REGION Network 4: Формирование событий линии
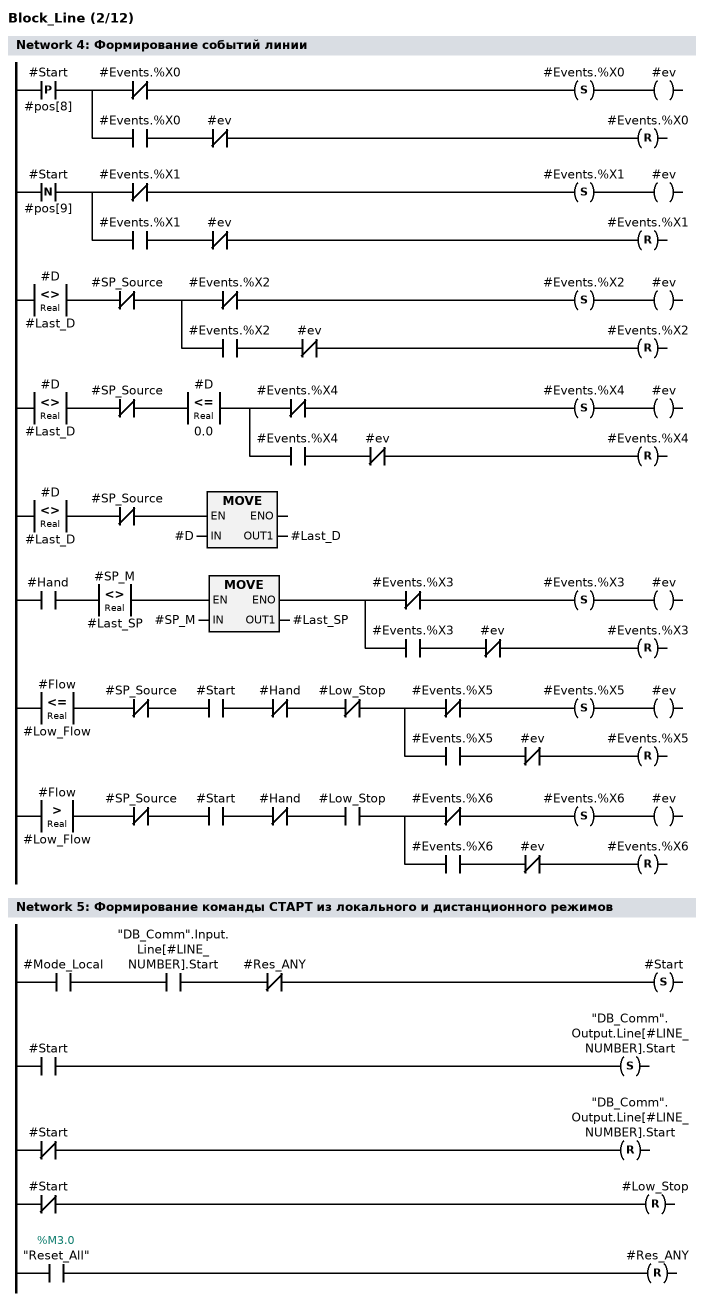
   RUNG wire#powerrail
      P_Contact(operand := #Start, bit := #pos[8])
      wire#w1
      I_Contact( #Events.%X0 )
      S_Coil( #Events.%X0 )
      Coil( #ev )
   END_RUNG
   RUNG wire#w1
      Contact( #Events.%X0 )
      I_Contact( #ev )
      R_Coil( #Events.%X0 )
   END_RUNG
   RUNG wire#powerrail
      N_Contact(operand := #Start, bit := #pos[9])
      wire#w2
      I_Contact( #Events.%X1 )
      S_Coil( #Events.%X1 )
      Coil( #ev )
   END_RUNG
   RUNG wire#w2
      Contact( #Events.%X1 )
      I_Contact( #ev )
      R_Coil( #Events.%X1 )
   END_RUNG
   RUNG wire#powerrail
      { S7_Templates := "SrcType := Real" } NE_Contact(in1 := #D, in2 := #Last_D)
      I_Contact( #SP_Source )
      wire#w3
      I_Contact( #Events.%X2 )
      S_Coil( #Events.%X2 )
      Coil( #ev )
   END_RUNG
   RUNG wire#w3
      Contact( #Events.%X2 )
      I_Contact( #ev )
      R_Coil( #Events.%X2 )
   END_RUNG
   RUNG wire#powerrail
      { S7_Templates := "SrcType := Real" } NE_Contact(in1 := #D, in2 := #Last_D)
      I_Contact( #SP_Source )
      { S7_Templates := "SrcType := Real" } LE_Contact(in1 := #D, in2 := 0.0)
      wire#w4
      I_Contact( #Events.%X4 )
      S_Coil( #Events.%X4 )
      Coil( #ev )
   END_RUNG
   RUNG wire#w4
      Contact( #Events.%X4 )
      I_Contact( #ev )
      R_Coil( #Events.%X4 )
   END_RUNG
   RUNG wire#powerrail
      { S7_Templates := "SrcType := Real" } NE_Contact(in1 := #D, in2 := #Last_D)
      I_Contact( #SP_Source )
      Move(in := #D, out1 => #Last_D)
   END_RUNG
   RUNG wire#powerrail
      Contact( #Hand )
      { S7_Templates := "SrcType := Real" } NE_Contact(in1 := #SP_M, in2 := #Last_SP)
      Move(in := #SP_M, out1 => #Last_SP)
      wire#w5
      I_Contact( #Events.%X3 )
      S_Coil( #Events.%X3 )
      Coil( #ev )
   END_RUNG
   RUNG wire#w5
      Contact( #Events.%X3 )
      I_Contact( #ev )
      R_Coil( #Events.%X3 )
   END_RUNG
   RUNG wire#powerrail
      { S7_Templates := "SrcType := Real" } LE_Contact(in1 := #Flow, in2 := #Low_Flow)
      I_Contact( #SP_Source )
      Contact( #Start )
      I_Contact( #Hand )
      I_Contact( #Low_Stop )
      wire#w6
      I_Contact( #Events.%X5 )
      S_Coil( #Events.%X5 )
      Coil( #ev )
   END_RUNG
   RUNG wire#w6
      Contact( #Events.%X5 )
      I_Contact( #ev )
      R_Coil( #Events.%X5 )
   END_RUNG
   RUNG wire#powerrail
      { S7_Templates := "SrcType := Real" } GT_Contact(in1 := #Flow, in2 := #Low_Flow)
      I_Contact( #SP_Source )
      Contact( #Start )
      I_Contact( #Hand )
      Contact( #Low_Stop )
      wire#w7
      I_Contact( #Events.%X6 )
      S_Coil( #Events.%X6 )
      Coil( #ev )
   END_RUNG
   RUNG wire#w7
      Contact( #Events.%X6 )
      I_Contact( #ev )
      R_Coil( #Events.%X6 )
   END_RUNG
   // the same network as SCL:
   #_w1 := #Start AND NOT #pos[8];   // rising edge of #Start
   #pos[8] := #Start;
   #_w2 := #_w1 AND NOT #Events.%X0;
   IF #_w2 THEN #Events.%X0 := TRUE; END_IF;
   #ev := #_w2;
   IF #_w1 AND #Events.%X0 AND NOT #ev THEN #Events.%X0 := FALSE; END_IF;
   #_w3 := NOT #Start AND #pos[9];   // falling edge of #Start
   #pos[9] := #Start;
   #_w4 := #_w3 AND NOT #Events.%X1;
   IF #_w4 THEN #Events.%X1 := TRUE; END_IF;
   #ev := #_w4;
   IF #_w3 AND #Events.%X1 AND NOT #ev THEN #Events.%X1 := FALSE; END_IF;
   #_w5 := (#D <> #Last_D) AND NOT #SP_Source;
   #_w6 := #_w5 AND NOT #Events.%X2;
   IF #_w6 THEN #Events.%X2 := TRUE; END_IF;
   #ev := #_w6;
   IF #_w5 AND #Events.%X2 AND NOT #ev THEN #Events.%X2 := FALSE; END_IF;
   #_w7 := (#D <> #Last_D) AND NOT #SP_Source AND (#D <= 0.0);
   #_w8 := #_w7 AND NOT #Events.%X4;
   IF #_w8 THEN #Events.%X4 := TRUE; END_IF;
   #ev := #_w8;
   IF #_w7 AND #Events.%X4 AND NOT #ev THEN #Events.%X4 := FALSE; END_IF;
   IF (#D <> #Last_D) AND NOT #SP_Source THEN #Last_D := #D; END_IF;
   #_w9 := #Hand AND (#SP_M <> #Last_SP);
   IF #_w9 THEN #Last_SP := #SP_M; END_IF;
   #_w10 := #_w9 AND NOT #Events.%X3;
   IF #_w10 THEN #Events.%X3 := TRUE; END_IF;
   #ev := #_w10;
   IF #_w9 AND #Events.%X3 AND NOT #ev THEN #Events.%X3 := FALSE; END_IF;
   #_w11 := (#Flow <= #Low_Flow) AND NOT #SP_Source AND #Start AND NOT #Hand AND NOT #Low_Stop;
   #_w12 := #_w11 AND NOT #Events.%X5;
   IF #_w12 THEN #Events.%X5 := TRUE; END_IF;
   #ev := #_w12;
   IF #_w11 AND #Events.%X5 AND NOT #ev THEN #Events.%X5 := FALSE; END_IF;
   #_w13 := (#Flow > #Low_Flow) AND NOT #SP_Source AND #Start AND NOT #Hand AND #Low_Stop;
   #_w14 := #_w13 AND NOT #Events.%X6;
   IF #_w14 THEN #Events.%X6 := TRUE; END_IF;
   #ev := #_w14;
   IF #_w13 AND #Events.%X6 AND NOT #ev THEN #Events.%X6 := FALSE; END_IF;
END_REGION

REGION Network 5: Формирование команды СТАРТ из локального и дистанционного режимов
   RUNG wire#powerrail
      Contact( #Mode_Local )
      Contact( "DB_Comm".Input.Line[#LINE_NUMBER].Start )
      I_Contact( #Res_ANY )
      S_Coil( #Start )
   END_RUNG
   RUNG wire#powerrail
      Contact( #Start )
      S_Coil( "DB_Comm".Output.Line[#LINE_NUMBER].Start )
   END_RUNG
   RUNG wire#powerrail
      I_Contact( #Start )
      R_Coil( "DB_Comm".Output.Line[#LINE_NUMBER].Start )
   END_RUNG
   RUNG wire#powerrail
      I_Contact( #Start )
      R_Coil( #Low_Stop )
   END_RUNG
   RUNG wire#powerrail
      Contact( "Reset_All" )
      R_Coil( #Res_ANY )
   END_RUNG
   // the same network as SCL:
   IF #Mode_Local AND "DB_Comm".Input.Line[#LINE_NUMBER].Start AND NOT #Res_ANY THEN #Start := TRUE; END_IF;
   IF #Start THEN "DB_Comm".Output.Line[#LINE_NUMBER].Start := TRUE; END_IF;
   IF NOT #Start THEN
       "DB_Comm".Output.Line[#LINE_NUMBER].Start := FALSE;
       #Low_Stop := FALSE;
   END_IF;
   IF "Reset_All" THEN #Res_ANY := FALSE; END_IF;
END_REGION

REGION Network 6: Старт - выбора насоса
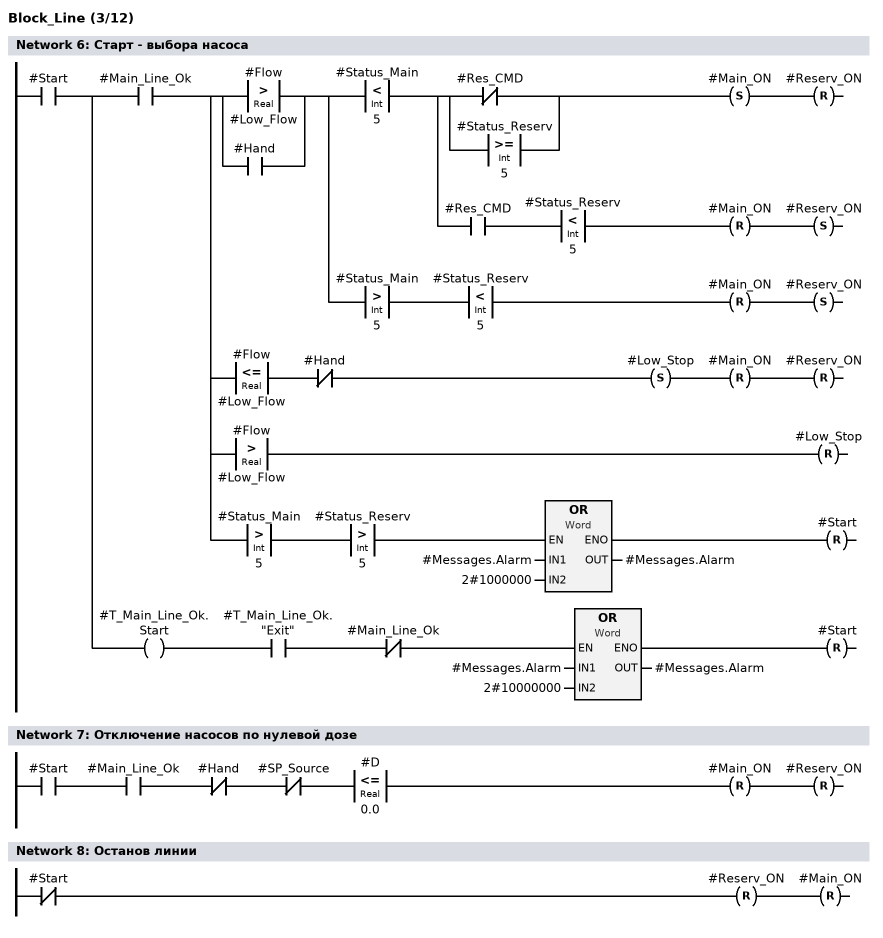
   #_w1 := #Start AND #Main_Line_Ok;
   #_w2 := #_w1 AND ((#Flow > #Low_Flow) OR #Hand);
   #_w3 := #_w2 AND (#Status_Main < 5);
   IF #_w3 AND (NOT #Res_CMD OR (#Status_Reserv >= 5)) THEN
       #Main_ON := TRUE;
       #Reserv_ON := FALSE;
   END_IF;
   IF #_w3 AND #Res_CMD AND (#Status_Reserv < 5) THEN
       #Main_ON := FALSE;
       #Reserv_ON := TRUE;
   END_IF;
   IF #_w2 AND (#Status_Main > 5) AND (#Status_Reserv < 5) THEN
       #Main_ON := FALSE;
       #Reserv_ON := TRUE;
   END_IF;
   IF #_w1 AND (#Flow <= #Low_Flow) AND NOT #Hand THEN
       #Low_Stop := TRUE;
       #Main_ON := FALSE;
       #Reserv_ON := FALSE;
   END_IF;
   IF #_w1 AND (#Flow > #Low_Flow) THEN #Low_Stop := FALSE; END_IF;
   IF #_w1 AND (#Status_Main > 5) AND (#Status_Reserv > 5) THEN
       #Messages.Alarm := #Messages.Alarm OR 2#1000000;
   END_IF;
   #_w4 := #Start;
   IF #_w1 AND (#Status_Main > 5) AND (#Status_Reserv > 5) THEN #Start := FALSE; END_IF;
   #T_Main_Line_Ok.Start := #_w4;
   IF #_w4 AND #T_Main_Line_Ok."Exit" AND NOT #Main_Line_Ok THEN
       #Messages.Alarm := #Messages.Alarm OR 2#10000000;
       #Start := FALSE;
   END_IF;
END_REGION

REGION Network 7: Отключение насосов по нулевой дозе
   RUNG wire#powerrail
      Contact( #Start )
      Contact( #Main_Line_Ok )
      I_Contact( #Hand )
      I_Contact( #SP_Source )
      { S7_Templates := "SrcType := Real" } LE_Contact(in1 := #D, in2 := 0.0)
      R_Coil( #Main_ON )
      R_Coil( #Reserv_ON )
   END_RUNG
   // the same network as SCL:
   IF #Start AND #Main_Line_Ok AND NOT #Hand AND NOT #SP_Source AND (#D <= 0.0) THEN
       #Main_ON := FALSE;
       #Reserv_ON := FALSE;
   END_IF;
END_REGION

REGION Network 8: Останов линии
   RUNG wire#powerrail
      I_Contact( #Start )
      R_Coil( #Reserv_ON )
      R_Coil( #Main_ON )
   END_RUNG
   // the same network as SCL:
   IF NOT #Start THEN
       #Reserv_ON := FALSE;
       #Main_ON := FALSE;
   END_IF;
END_REGION

REGION Network 9: Подсчёт наработки насосов и управление выбором основного и резервного
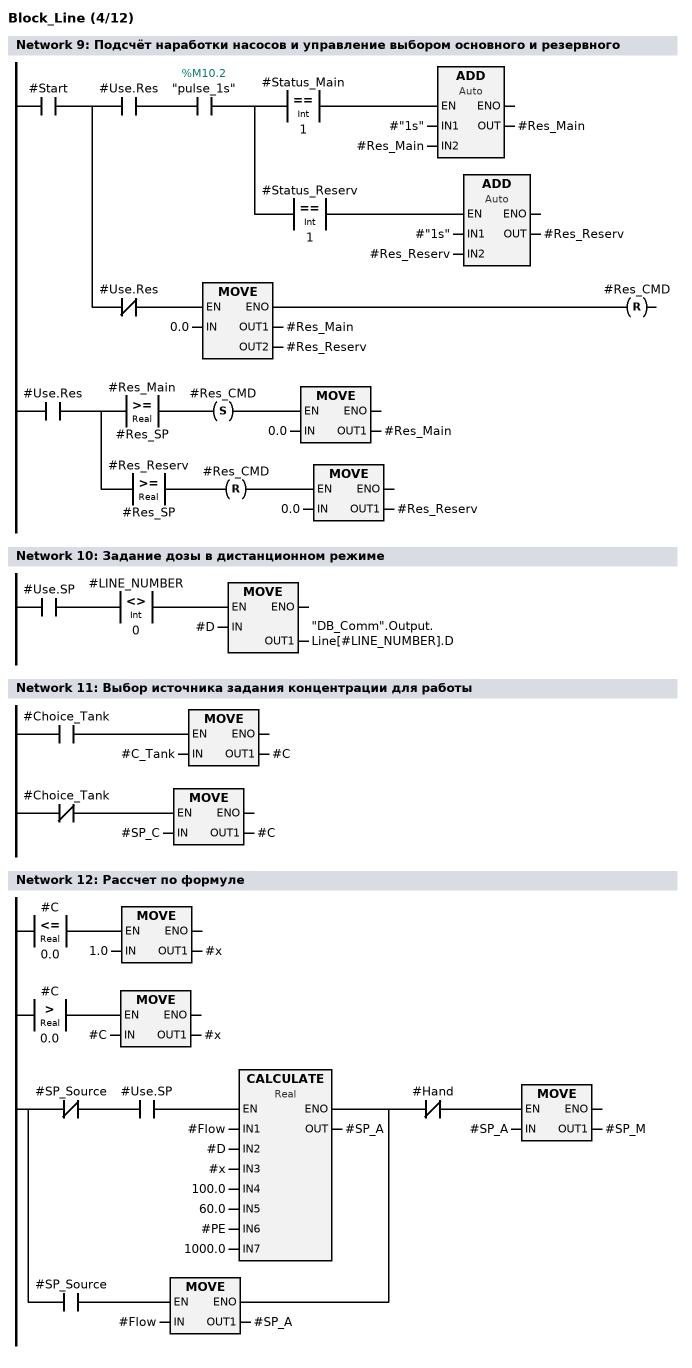
   RUNG wire#powerrail
      Contact( #Start )
      wire#w1
      Contact( #Use.Res )
      Contact( "pulse_1s" )
      wire#w2
      { S7_Templates := "SrcType := Int" } EQ_Contact(in1 := #Status_Main, in2 := 1)
      Add(in1 := #"1s", in2 := #Res_Main, out => #Res_Main)
   END_RUNG
   RUNG wire#w2
      { S7_Templates := "SrcType := Int" } EQ_Contact(in1 := #Status_Reserv, in2 := 1)
      Add(in1 := #"1s", in2 := #Res_Reserv, out => #Res_Reserv)
   END_RUNG
   RUNG wire#w1
      I_Contact( #Use.Res )
      Move(in := 0.0, out1 => #Res_Main, out2 => #Res_Reserv)
      R_Coil( #Res_CMD )
   END_RUNG
   RUNG wire#powerrail
      Contact( #Use.Res )
      wire#w3
      { S7_Templates := "SrcType := Real" } GE_Contact(in1 := #Res_Main, in2 := #Res_SP)
      S_Coil( #Res_CMD )
      Move(in := 0.0, out1 => #Res_Main)
   END_RUNG
   RUNG wire#w3
      { S7_Templates := "SrcType := Real" } GE_Contact(in1 := #Res_Reserv, in2 := #Res_SP)
      R_Coil( #Res_CMD )
      Move(in := 0.0, out1 => #Res_Reserv)
   END_RUNG
   // the same network as SCL:
   #_w1 := #Start AND #Use.Res AND "pulse_1s";
   IF #_w1 AND (#Status_Main = 1) THEN #Res_Main := #"1s" + #Res_Main; END_IF;
   IF #_w1 AND (#Status_Reserv = 1) THEN #Res_Reserv := #"1s" + #Res_Reserv; END_IF;
   IF #Start AND NOT #Use.Res THEN
       #Res_Main := 0.0;
       #Res_Reserv := 0.0;
       #Res_CMD := FALSE;
   END_IF;
   IF #Use.Res AND (#Res_Main >= #Res_SP) THEN
       #Res_CMD := TRUE;
       #Res_Main := 0.0;
   END_IF;
   IF #Use.Res AND (#Res_Reserv >= #Res_SP) THEN
       #Res_CMD := FALSE;
       #Res_Reserv := 0.0;
   END_IF;
END_REGION

REGION Network 10: Задание дозы в дистанционном режиме
   RUNG wire#powerrail
      Contact( #Use.SP )
      { S7_Templates := "SrcType := Int" } NE_Contact(in1 := #LINE_NUMBER, in2 := 0)
      Move(in := #D, out1 => "DB_Comm".Output.Line[#LINE_NUMBER].D)
   END_RUNG
   // the same network as SCL:
   IF #Use.SP AND (#LINE_NUMBER <> 0) THEN "DB_Comm".Output.Line[#LINE_NUMBER].D := #D; END_IF;
END_REGION

REGION Network 11: Выбор источника задания концентрации для работы
   RUNG wire#powerrail
      Contact( #Choice_Tank )
      Move(in := #C_Tank, out1 => #C)
   END_RUNG
   RUNG wire#powerrail
      I_Contact( #Choice_Tank )
      Move(in := #SP_C, out1 => #C)
   END_RUNG
   // the same network as SCL:
   IF #Choice_Tank THEN #C := #C_Tank; END_IF;
   IF NOT #Choice_Tank THEN #C := #SP_C; END_IF;
END_REGION

REGION Network 12: Рассчет по формуле
   RUNG wire#powerrail
      { S7_Templates := "SrcType := Real" } LE_Contact(in1 := #C, in2 := 0.0)
      Move(in := 1.0, out1 => #x)
   END_RUNG
   RUNG wire#powerrail
      { S7_Templates := "SrcType := Real" } GT_Contact(in1 := #C, in2 := 0.0)
      Move(in := #C, out1 => #x)
   END_RUNG
   RUNG wire#powerrail
      I_Contact( #SP_Source )
      Contact( #Use.SP )
      { S7_Templates := "SrcType := Real"; S7_Expression := "(IN2 * IN1) / ( IN3 / IN4) / (IN6 * IN7) / IN5" } Calculate(in1 := #Flow, in2 := #D, in3 := #x, in4 := 100.0, in5 := 60.0, in6 := #PE, in7 := 1000.0, out => #SP_A)
      wire#w1
      I_Contact( #Hand )
      Move(in := #SP_A, out1 => #SP_M)
   END_RUNG
   RUNG wire#powerrail
      Contact( #SP_Source )
      Move(in := #Flow, out1 => #SP_A)
   END_RUNG wire#w1
   // the same network as SCL:
   IF #C <= 0.0 THEN #x := 1.0; END_IF;
   IF #C > 0.0 THEN #x := #C; END_IF;
   #_w1 := NOT #SP_Source AND #Use.SP;
   IF #_w1 THEN #SP_A := (#D * #Flow) / ( #x / 100.0) / (#PE * 1000.0) / 60.0; END_IF;
   IF #SP_Source THEN #SP_A := #Flow; END_IF;
   IF (#_w1 OR #SP_Source) AND NOT #Hand THEN #SP_M := #SP_A; END_IF;
END_REGION

REGION Network 13: Выбор режима с разбавлением или без разбавления в дистанционном режиме
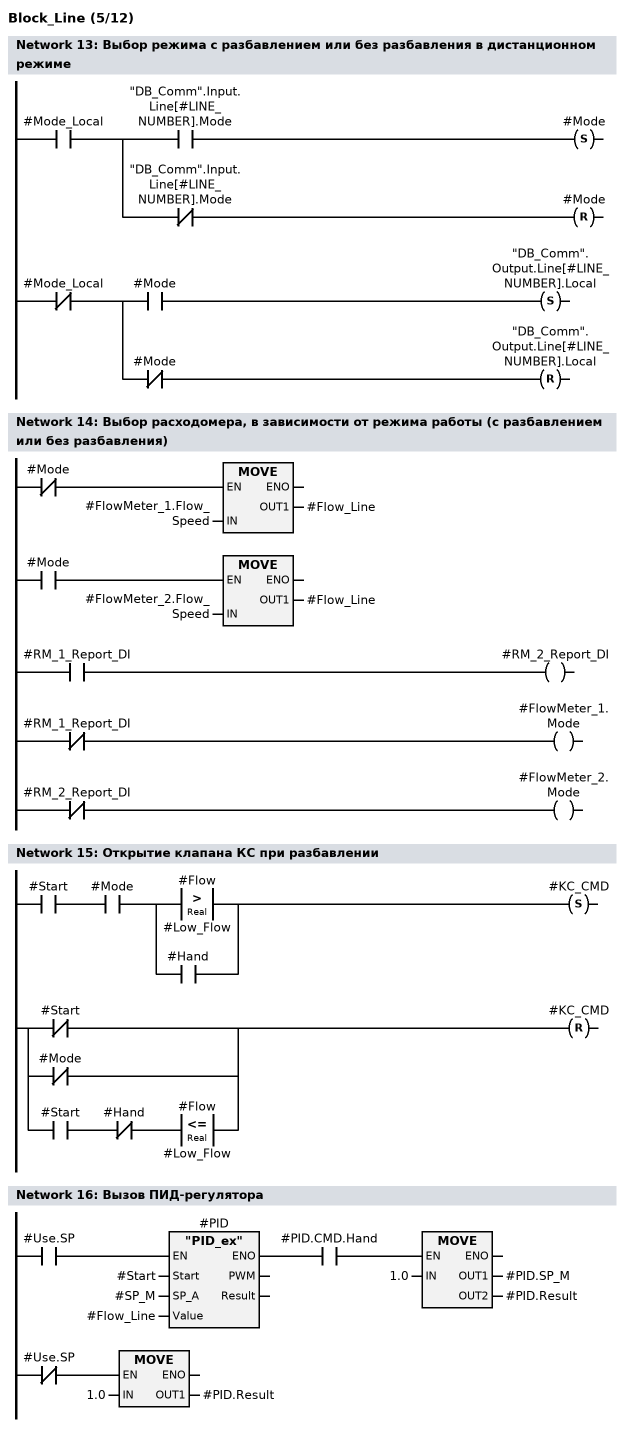
   RUNG wire#powerrail
      Contact( #Mode_Local )
      wire#w1
      Contact( "DB_Comm".Input.Line[#LINE_NUMBER].Mode )
      S_Coil( #Mode )
   END_RUNG
   RUNG wire#w1
      I_Contact( "DB_Comm".Input.Line[#LINE_NUMBER].Mode )
      R_Coil( #Mode )
   END_RUNG
   RUNG wire#powerrail
      I_Contact( #Mode_Local )
      wire#w2
      Contact( #Mode )
      S_Coil( "DB_Comm".Output.Line[#LINE_NUMBER].Local )
   END_RUNG
   RUNG wire#w2
      I_Contact( #Mode )
      R_Coil( "DB_Comm".Output.Line[#LINE_NUMBER].Local )
   END_RUNG
   // the same network as SCL:
   IF #Mode_Local AND "DB_Comm".Input.Line[#LINE_NUMBER].Mode THEN #Mode := TRUE; END_IF;
   IF #Mode_Local AND NOT "DB_Comm".Input.Line[#LINE_NUMBER].Mode THEN #Mode := FALSE; END_IF;
   IF NOT #Mode_Local AND #Mode THEN "DB_Comm".Output.Line[#LINE_NUMBER].Local := TRUE; END_IF;
   IF NOT #Mode_Local AND NOT #Mode THEN "DB_Comm".Output.Line[#LINE_NUMBER].Local := FALSE; END_IF;
END_REGION

REGION Network 14: Выбор расходомера, в зависимости от режима работы (с разбавлением или без разбавления)
   RUNG wire#powerrail
      I_Contact( #Mode )
      Move(in := #FlowMeter_1.Flow_Speed, out1 => #Flow_Line)
   END_RUNG
   RUNG wire#powerrail
      Contact( #Mode )
      Move(in := #FlowMeter_2.Flow_Speed, out1 => #Flow_Line)
   END_RUNG
   RUNG wire#powerrail
      Contact( #RM_1_Report_DI )
      Coil( #RM_2_Report_DI )
   END_RUNG
   RUNG wire#powerrail
      I_Contact( #RM_1_Report_DI )
      Coil( #FlowMeter_1.Mode )
   END_RUNG
   RUNG wire#powerrail
      I_Contact( #RM_2_Report_DI )
      Coil( #FlowMeter_2.Mode )
   END_RUNG
   // the same network as SCL:
   IF NOT #Mode THEN #Flow_Line := #FlowMeter_1.Flow_Speed; END_IF;
   IF #Mode THEN #Flow_Line := #FlowMeter_2.Flow_Speed; END_IF;
   #RM_2_Report_DI := #RM_1_Report_DI;
   #FlowMeter_1.Mode := NOT #RM_1_Report_DI;
   #FlowMeter_2.Mode := NOT #RM_2_Report_DI;
END_REGION

REGION Network 15: Открытие клапана КС при разбавлении
   RUNG wire#powerrail
      Contact( #Start )
      Contact( #Mode )
      wire#w1
      { S7_Templates := "SrcType := Real" } GT_Contact(in1 := #Flow, in2 := #Low_Flow)
      wire#w2
      S_Coil( #KC_CMD )
   END_RUNG
   RUNG wire#w1
      Contact( #Hand )
   END_RUNG wire#w2
   RUNG wire#powerrail
      I_Contact( #Start )
      wire#w3
      R_Coil( #KC_CMD )
   END_RUNG
   RUNG wire#powerrail
      I_Contact( #Mode )
   END_RUNG wire#w3
   RUNG wire#powerrail
      Contact( #Start )
      I_Contact( #Hand )
      { S7_Templates := "SrcType := Real" } LE_Contact(in1 := #Flow, in2 := #Low_Flow)
   END_RUNG wire#w3
   // the same network as SCL:
   IF #Start AND #Mode AND ((#Flow > #Low_Flow) OR #Hand) THEN #KC_CMD := TRUE; END_IF;
   IF NOT #Start OR NOT #Mode OR (#Start AND NOT #Hand AND (#Flow <= #Low_Flow)) THEN
       #KC_CMD := FALSE;
   END_IF;
END_REGION

REGION Network 16: Вызов ПИД-регулятора
   RUNG wire#powerrail
      Contact( #Use.SP )
      #PID(Start := #Start, SP_A := #SP_M, Value := #Flow_Line, PWM =>, Result =>)
      Contact( #PID.CMD.Hand )
      Move(in := 1.0, out1 => #PID.SP_M, out2 => #PID.Result)
   END_RUNG
   RUNG wire#powerrail
      I_Contact( #Use.SP )
      Move(in := 1.0, out1 => #PID.Result)
   END_RUNG
   // the same network as SCL:
   #PID(EN := #Use.SP, Start := #Start, SP_A := #SP_M, Value := #Flow_Line, ENO => #_w1);   // "PID_ex"
   IF #_w1 AND #PID.CMD.Hand THEN
       #PID.SP_M := 1.0;
       #PID.Result := 1.0;
   END_IF;
   IF NOT #Use.SP THEN #PID.Result := 1.0; END_IF;
END_REGION

REGION Network 17: Обнуление уставки при отстутствии аналогового управления насосами
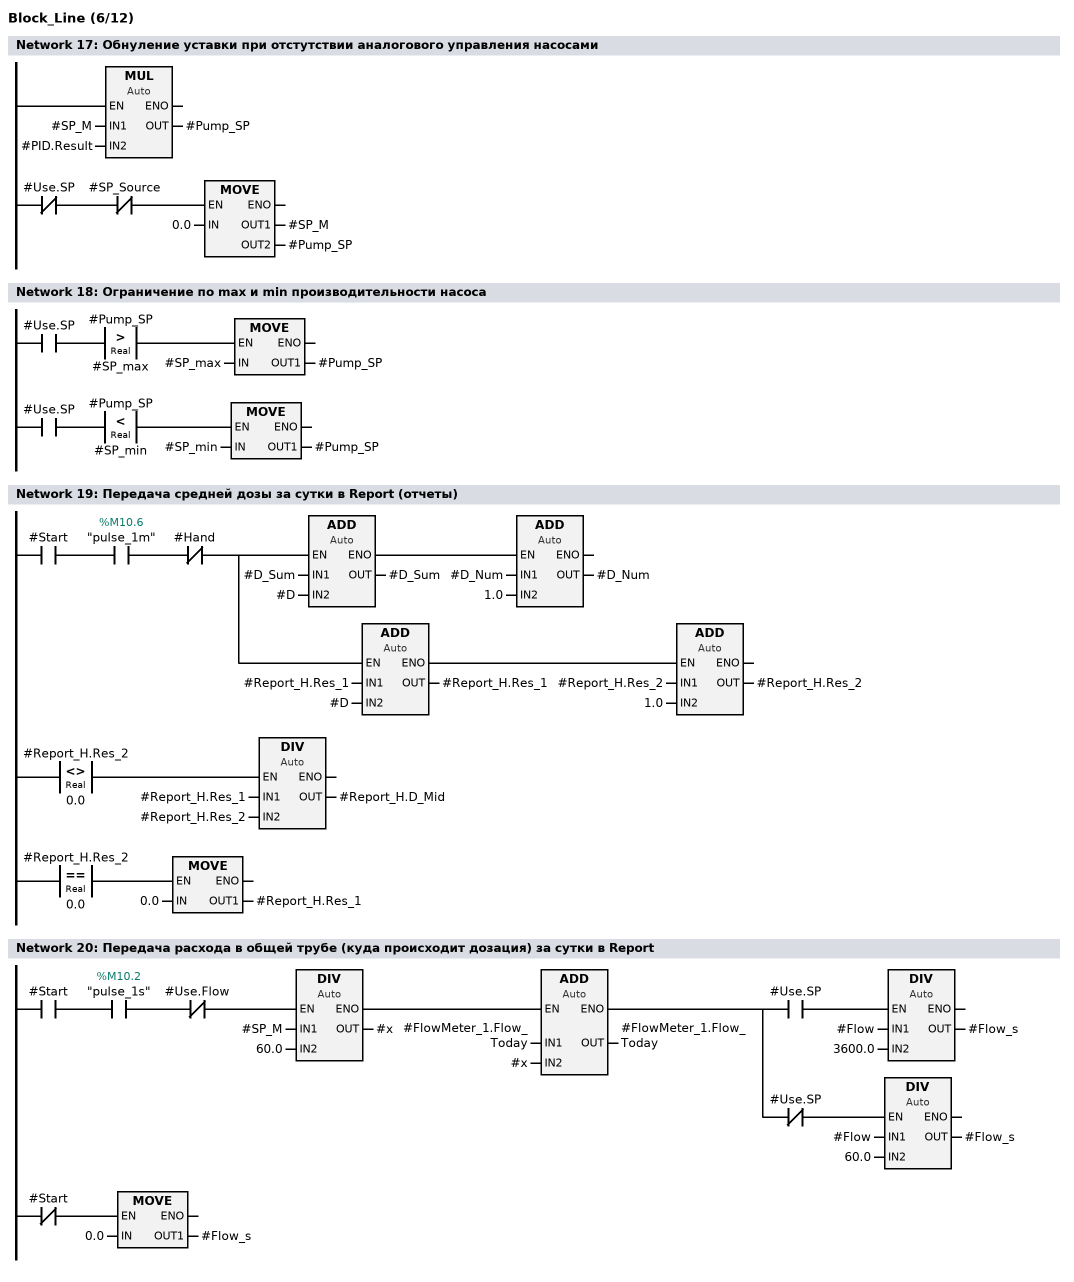
   RUNG wire#powerrail
      Mul(in1 := #SP_M, in2 := #PID.Result, out => #Pump_SP)
   END_RUNG
   RUNG wire#powerrail
      I_Contact( #Use.SP )
      I_Contact( #SP_Source )
      Move(in := 0.0, out1 => #SP_M, out2 => #Pump_SP)
   END_RUNG
   // the same network as SCL:
   #Pump_SP := #SP_M * #PID.Result;
   IF NOT #Use.SP AND NOT #SP_Source THEN
       #SP_M := 0.0;
       #Pump_SP := 0.0;
   END_IF;
END_REGION

REGION Network 18: Ограничение по max и min производительности насоса
   RUNG wire#powerrail
      Contact( #Use.SP )
      { S7_Templates := "SrcType := Real" } GT_Contact(in1 := #Pump_SP, in2 := #SP_max)
      Move(in := #SP_max, out1 => #Pump_SP)
   END_RUNG
   RUNG wire#powerrail
      Contact( #Use.SP )
      { S7_Templates := "SrcType := Real" } LT_Contact(in1 := #Pump_SP, in2 := #SP_min)
      Move(in := #SP_min, out1 => #Pump_SP)
   END_RUNG
   // the same network as SCL:
   IF #Use.SP AND (#Pump_SP > #SP_max) THEN #Pump_SP := #SP_max; END_IF;
   IF #Use.SP AND (#Pump_SP < #SP_min) THEN #Pump_SP := #SP_min; END_IF;
END_REGION

REGION Network 19: Передача средней дозы за сутки в Report (отчеты)
   RUNG wire#powerrail
      Contact( #Start )
      Contact( "pulse_1m" )
      I_Contact( #Hand )
      wire#w1
      Add(in1 := #D_Sum, in2 := #D, out => #D_Sum)
      Add(in1 := #D_Num, in2 := 1.0, out => #D_Num)
   END_RUNG
   RUNG wire#w1
      Add(in1 := #Report_H.Res_1, in2 := #D, out => #Report_H.Res_1)
      Add(in1 := #Report_H.Res_2, in2 := 1.0, out => #Report_H.Res_2)
   END_RUNG
   RUNG wire#powerrail
      { S7_Templates := "SrcType := Real" } NE_Contact(in1 := #Report_H.Res_2, in2 := 0.0)
      Div(in1 := #Report_H.Res_1, in2 := #Report_H.Res_2, out => #Report_H.D_Mid)
   END_RUNG
   RUNG wire#powerrail
      { S7_Templates := "SrcType := Real" } EQ_Contact(in1 := #Report_H.Res_2, in2 := 0.0)
      Move(in := 0.0, out1 => #Report_H.Res_1)
   END_RUNG
   // the same network as SCL:
   IF #Start AND "pulse_1m" AND NOT #Hand THEN
       #D_Sum := #D_Sum + #D;
       #D_Num := #D_Num + 1.0;
       #Report_H.Res_1 := #Report_H.Res_1 + #D;
       #Report_H.Res_2 := #Report_H.Res_2 + 1.0;
   END_IF;
   IF #Report_H.Res_2 <> 0.0 THEN #Report_H.D_Mid := #Report_H.Res_1 / #Report_H.Res_2; END_IF;
   IF #Report_H.Res_2 = 0.0 THEN #Report_H.Res_1 := 0.0; END_IF;
END_REGION

REGION Network 20: Передача расхода в общей трубе (куда происходит дозация) за сутки в Report
   RUNG wire#powerrail
      Contact( #Start )
      Contact( "pulse_1s" )
      I_Contact( #Use.Flow )
      Div(in1 := #SP_M, in2 := 60.0, out => #x)
      Add(in1 := #FlowMeter_1.Flow_Today, in2 := #x, out => #FlowMeter_1.Flow_Today)
      wire#w1
      Contact( #Use.SP )
      Div(in1 := #Flow, in2 := 3600.0, out => #Flow_s)
   END_RUNG
   RUNG wire#w1
      I_Contact( #Use.SP )
      Div(in1 := #Flow, in2 := 60.0, out => #Flow_s)
   END_RUNG
   RUNG wire#powerrail
      I_Contact( #Start )
      Move(in := 0.0, out1 => #Flow_s)
   END_RUNG
   // the same network as SCL:
   #_w1 := #Start AND "pulse_1s" AND NOT #Use.Flow;
   IF #_w1 THEN
       #x := #SP_M / 60.0;
       #FlowMeter_1.Flow_Today := #FlowMeter_1.Flow_Today + #x;
   END_IF;
   IF #_w1 AND #Use.SP THEN #Flow_s := #Flow / 3600.0; END_IF;
   IF #_w1 AND NOT #Use.SP THEN #Flow_s := #Flow / 60.0; END_IF;
   IF NOT #Start THEN #Flow_s := 0.0; END_IF;
END_REGION

REGION Network 21: Авария основного насоса по датчику протока
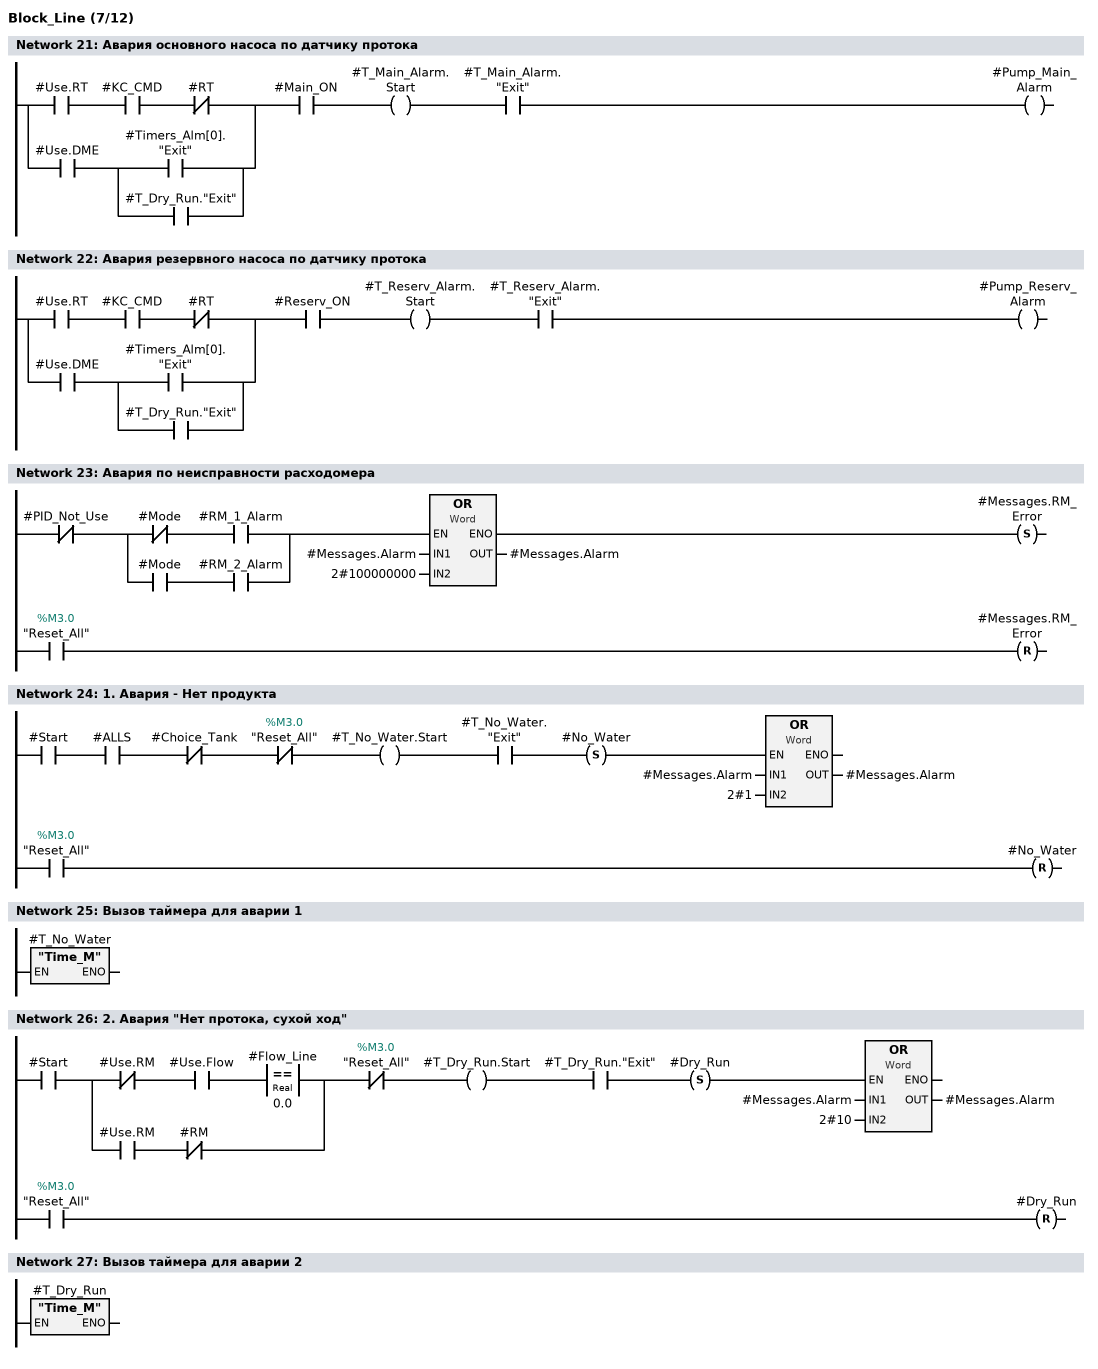
   RUNG wire#powerrail
      Contact( #Use.RT )
      Contact( #KC_CMD )
      I_Contact( #RT )
      wire#w1
      Contact( #Main_ON )
      Coil( #T_Main_Alarm.Start )
      Contact( #T_Main_Alarm."Exit" )
      Coil( #Pump_Main_Alarm )
   END_RUNG
   RUNG wire#powerrail
      Contact( #Use.DME )
      wire#w2
      Contact( #Timers_Alm[0]."Exit" )
   END_RUNG wire#w1
   RUNG wire#w2
      Contact( #T_Dry_Run."Exit" )
   END_RUNG wire#w1
   // the same network as SCL:
   #T_Main_Alarm.Start := ((#Use.RT AND #KC_CMD AND NOT #RT) OR (#Use.DME AND (#Timers_Alm[0]."Exit" OR #T_Dry_Run."Exit"))) AND #Main_ON;
   #Pump_Main_Alarm := #T_Main_Alarm.Start AND #T_Main_Alarm."Exit";
END_REGION

REGION Network 22: Авария резервного насоса по датчику протока
   RUNG wire#powerrail
      Contact( #Use.RT )
      Contact( #KC_CMD )
      I_Contact( #RT )
      wire#w1
      Contact( #Reserv_ON )
      Coil( #T_Reserv_Alarm.Start )
      Contact( #T_Reserv_Alarm."Exit" )
      Coil( #Pump_Reserv_Alarm )
   END_RUNG
   RUNG wire#powerrail
      Contact( #Use.DME )
      wire#w2
      Contact( #Timers_Alm[0]."Exit" )
   END_RUNG wire#w1
   RUNG wire#w2
      Contact( #T_Dry_Run."Exit" )
   END_RUNG wire#w1
   // the same network as SCL:
   #T_Reserv_Alarm.Start := ((#Use.RT AND #KC_CMD AND NOT #RT) OR (#Use.DME AND (#Timers_Alm[0]."Exit" OR #T_Dry_Run."Exit"))) AND #Reserv_ON;
   #Pump_Reserv_Alarm := #T_Reserv_Alarm.Start AND #T_Reserv_Alarm."Exit";
END_REGION

REGION Network 23: Авария по неисправности расходомера
   IF NOT #PID_Not_Use AND ((NOT #Mode AND #RM_1_Alarm) OR (#Mode AND #RM_2_Alarm)) THEN
       #Messages.Alarm := #Messages.Alarm OR 2#100000000;
       #Messages.RM_Error := TRUE;
   END_IF;
   IF "Reset_All" THEN #Messages.RM_Error := FALSE; END_IF;
END_REGION

REGION Network 24: 1. Авария - Нет продукта
   #T_No_Water.Start := #Start AND #ALLS AND NOT #Choice_Tank AND NOT "Reset_All";
   IF #T_No_Water.Start AND #T_No_Water."Exit" THEN
       #No_Water := TRUE;
       #Messages.Alarm := #Messages.Alarm OR 2#1;
   END_IF;
   IF "Reset_All" THEN #No_Water := FALSE; END_IF;
END_REGION

REGION Network 25: Вызов таймера для аварии 1
   RUNG wire#powerrail
      #T_No_Water()
   END_RUNG
   // the same network as SCL:
   #T_No_Water();   // "Time_M"
END_REGION

REGION Network 26: 2. Авария "Нет протока, сухой ход"
   #T_Dry_Run.Start := #Start AND ((NOT #Use.RM AND #Use.Flow AND (#Flow_Line = 0.0)) OR (#Use.RM AND NOT #RM)) AND NOT "Reset_All";
   IF #T_Dry_Run.Start AND #T_Dry_Run."Exit" THEN
       #Dry_Run := TRUE;
       #Messages.Alarm := #Messages.Alarm OR 2#10;
   END_IF;
   IF "Reset_All" THEN #Dry_Run := FALSE; END_IF;
END_REGION

REGION Network 27: Вызов таймера для аварии 2
   RUNG wire#powerrail
      #T_Dry_Run()
   END_RUNG
   // the same network as SCL:
   #T_Dry_Run();   // "Time_M"
END_REGION

REGION Network 28: 3. Авария - низкий проток
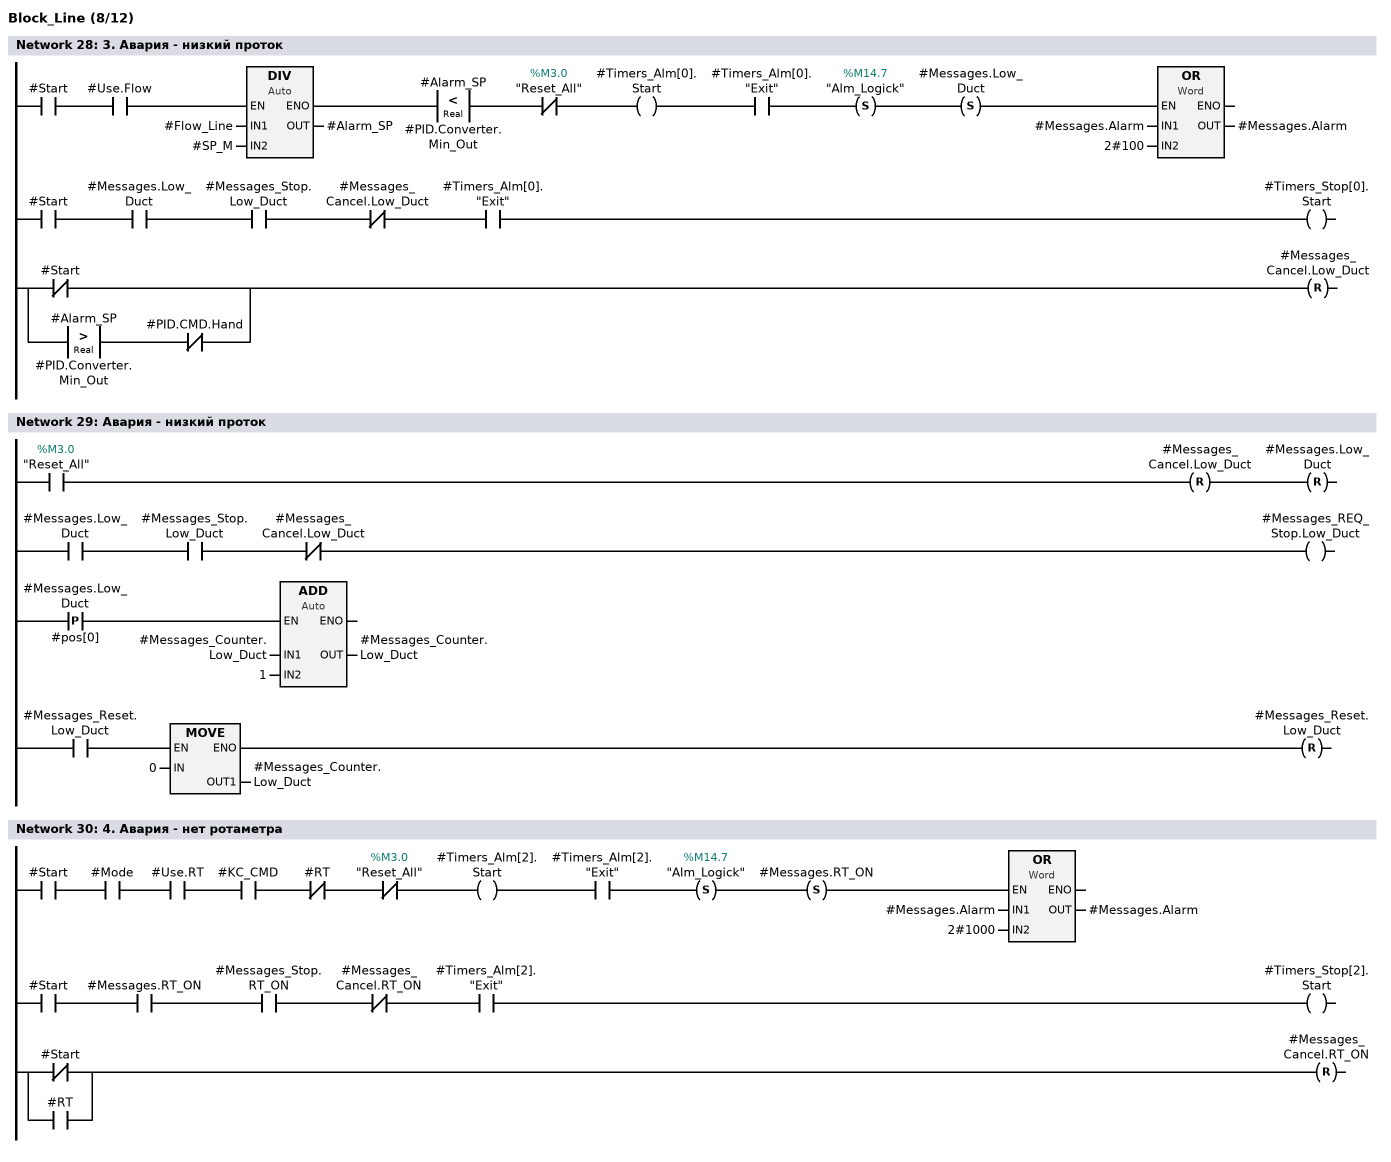
   #_w1 := #Start AND #Use.Flow;
   IF #_w1 THEN #Alarm_SP := #Flow_Line / #SP_M; END_IF;
   #Timers_Alm[0].Start := #_w1 AND (#Alarm_SP < #PID.Converter.Min_Out) AND NOT "Reset_All";
   IF #_w1 AND (#Alarm_SP < #PID.Converter.Min_Out) AND NOT "Reset_All" AND #Timers_Alm[0]."Exit" THEN
       "Alm_Logick" := TRUE;
       #Messages.Low_Duct := TRUE;
       #Messages.Alarm := #Messages.Alarm OR 2#100;
   END_IF;
   #Timers_Stop[0].Start := #Start AND #Messages.Low_Duct AND #Messages_Stop.Low_Duct AND NOT #Messages_Cancel.Low_Duct AND #Timers_Alm[0]."Exit";
   IF NOT #Start OR ((#Alarm_SP > #PID.Converter.Min_Out) AND NOT #PID.CMD.Hand) THEN
       #Messages_Cancel.Low_Duct := FALSE;
   END_IF;
END_REGION

REGION Network 29: Авария - низкий проток
   RUNG wire#powerrail
      Contact( "Reset_All" )
      R_Coil( #Messages_Cancel.Low_Duct )
      R_Coil( #Messages.Low_Duct )
   END_RUNG
   RUNG wire#powerrail
      Contact( #Messages.Low_Duct )
      Contact( #Messages_Stop.Low_Duct )
      I_Contact( #Messages_Cancel.Low_Duct )
      Coil( #Messages_REQ_Stop.Low_Duct )
   END_RUNG
   RUNG wire#powerrail
      P_Contact(operand := #Messages.Low_Duct, bit := #pos[0])
      Add(in1 := #Messages_Counter.Low_Duct, in2 := 1, out => #Messages_Counter.Low_Duct)
   END_RUNG
   RUNG wire#powerrail
      Contact( #Messages_Reset.Low_Duct )
      Move(in := 0, out1 => #Messages_Counter.Low_Duct)
      R_Coil( #Messages_Reset.Low_Duct )
   END_RUNG
   // the same network as SCL:
   IF "Reset_All" THEN
       #Messages_Cancel.Low_Duct := FALSE;
       #Messages.Low_Duct := FALSE;
   END_IF;
   #Messages_REQ_Stop.Low_Duct := #Messages.Low_Duct AND #Messages_Stop.Low_Duct AND NOT #Messages_Cancel.Low_Duct;
   #_w1 := #Messages.Low_Duct AND NOT #pos[0];   // rising edge of #Messages.Low_Duct
   #pos[0] := #Messages.Low_Duct;
   IF #_w1 THEN #Messages_Counter.Low_Duct := #Messages_Counter.Low_Duct + 1; END_IF;
   IF #Messages_Reset.Low_Duct THEN
       #Messages_Counter.Low_Duct := 0;
       #Messages_Reset.Low_Duct := FALSE;
   END_IF;
END_REGION

REGION Network 30: 4. Авария - нет ротаметра
   #Timers_Alm[2].Start := #Start AND #Mode AND #Use.RT AND #KC_CMD AND NOT #RT AND NOT "Reset_All";
   IF #Start AND #Mode AND #Use.RT AND #KC_CMD AND NOT #RT AND NOT "Reset_All" AND #Timers_Alm[2]."Exit" THEN
       "Alm_Logick" := TRUE;
       #Messages.RT_ON := TRUE;
       #Messages.Alarm := #Messages.Alarm OR 2#1000;
   END_IF;
   #Timers_Stop[2].Start := #Start AND #Messages.RT_ON AND #Messages_Stop.RT_ON AND NOT #Messages_Cancel.RT_ON AND #Timers_Alm[2]."Exit";
   IF NOT #Start OR #RT THEN #Messages_Cancel.RT_ON := FALSE; END_IF;
END_REGION

REGION Network 31: Авария - нет ротаметра
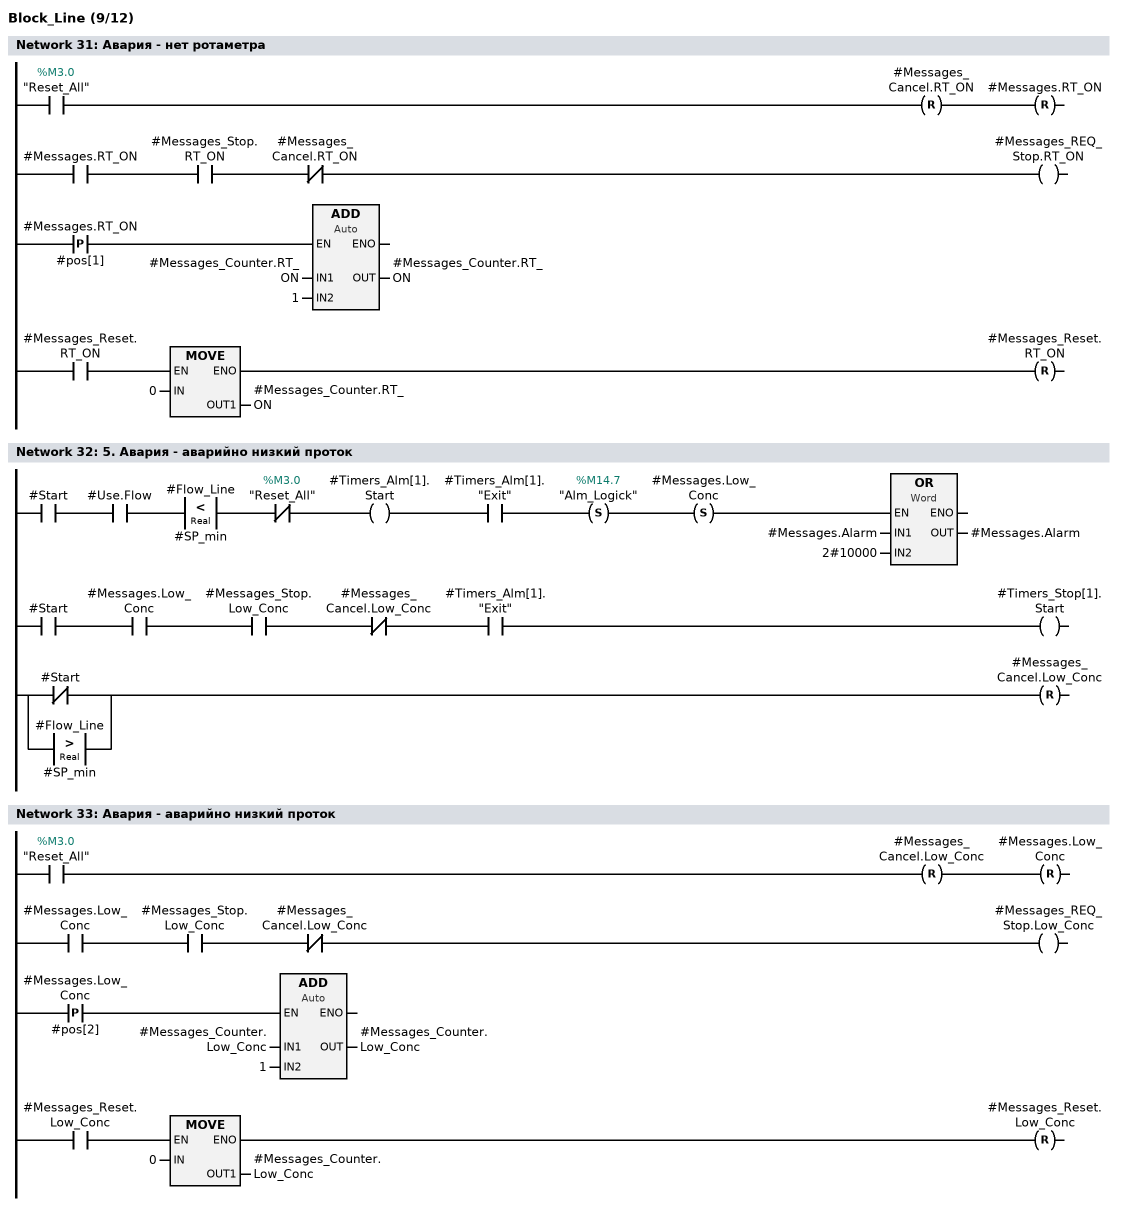
   RUNG wire#powerrail
      Contact( "Reset_All" )
      R_Coil( #Messages_Cancel.RT_ON )
      R_Coil( #Messages.RT_ON )
   END_RUNG
   RUNG wire#powerrail
      Contact( #Messages.RT_ON )
      Contact( #Messages_Stop.RT_ON )
      I_Contact( #Messages_Cancel.RT_ON )
      Coil( #Messages_REQ_Stop.RT_ON )
   END_RUNG
   RUNG wire#powerrail
      P_Contact(operand := #Messages.RT_ON, bit := #pos[1])
      Add(in1 := #Messages_Counter.RT_ON, in2 := 1, out => #Messages_Counter.RT_ON)
   END_RUNG
   RUNG wire#powerrail
      Contact( #Messages_Reset.RT_ON )
      Move(in := 0, out1 => #Messages_Counter.RT_ON)
      R_Coil( #Messages_Reset.RT_ON )
   END_RUNG
   // the same network as SCL:
   IF "Reset_All" THEN
       #Messages_Cancel.RT_ON := FALSE;
       #Messages.RT_ON := FALSE;
   END_IF;
   #Messages_REQ_Stop.RT_ON := #Messages.RT_ON AND #Messages_Stop.RT_ON AND NOT #Messages_Cancel.RT_ON;
   #_w1 := #Messages.RT_ON AND NOT #pos[1];   // rising edge of #Messages.RT_ON
   #pos[1] := #Messages.RT_ON;
   IF #_w1 THEN #Messages_Counter.RT_ON := #Messages_Counter.RT_ON + 1; END_IF;
   IF #Messages_Reset.RT_ON THEN
       #Messages_Counter.RT_ON := 0;
       #Messages_Reset.RT_ON := FALSE;
   END_IF;
END_REGION

REGION Network 32: 5. Авария - аварийно низкий проток
   #Timers_Alm[1].Start := #Start AND #Use.Flow AND (#Flow_Line < #SP_min) AND NOT "Reset_All";
   IF #Start AND #Use.Flow AND (#Flow_Line < #SP_min) AND NOT "Reset_All" AND #Timers_Alm[1]."Exit" THEN
       "Alm_Logick" := TRUE;
       #Messages.Low_Conc := TRUE;
       #Messages.Alarm := #Messages.Alarm OR 2#10000;
   END_IF;
   #Timers_Stop[1].Start := #Start AND #Messages.Low_Conc AND #Messages_Stop.Low_Conc AND NOT #Messages_Cancel.Low_Conc AND #Timers_Alm[1]."Exit";
   IF NOT #Start OR (#Flow_Line > #SP_min) THEN #Messages_Cancel.Low_Conc := FALSE; END_IF;
END_REGION

REGION Network 33: Авария - аварийно низкий проток
   RUNG wire#powerrail
      Contact( "Reset_All" )
      R_Coil( #Messages_Cancel.Low_Conc )
      R_Coil( #Messages.Low_Conc )
   END_RUNG
   RUNG wire#powerrail
      Contact( #Messages.Low_Conc )
      Contact( #Messages_Stop.Low_Conc )
      I_Contact( #Messages_Cancel.Low_Conc )
      Coil( #Messages_REQ_Stop.Low_Conc )
   END_RUNG
   RUNG wire#powerrail
      P_Contact(operand := #Messages.Low_Conc, bit := #pos[2])
      Add(in1 := #Messages_Counter.Low_Conc, in2 := 1, out => #Messages_Counter.Low_Conc)
   END_RUNG
   RUNG wire#powerrail
      Contact( #Messages_Reset.Low_Conc )
      Move(in := 0, out1 => #Messages_Counter.Low_Conc)
      R_Coil( #Messages_Reset.Low_Conc )
   END_RUNG
   // the same network as SCL:
   IF "Reset_All" THEN
       #Messages_Cancel.Low_Conc := FALSE;
       #Messages.Low_Conc := FALSE;
   END_IF;
   #Messages_REQ_Stop.Low_Conc := #Messages.Low_Conc AND #Messages_Stop.Low_Conc AND NOT #Messages_Cancel.Low_Conc;
   #_w1 := #Messages.Low_Conc AND NOT #pos[2];   // rising edge of #Messages.Low_Conc
   #pos[2] := #Messages.Low_Conc;
   IF #_w1 THEN #Messages_Counter.Low_Conc := #Messages_Counter.Low_Conc + 1; END_IF;
   IF #Messages_Reset.Low_Conc THEN
       #Messages_Counter.Low_Conc := 0;
       #Messages_Reset.Low_Conc := FALSE;
   END_IF;
END_REGION

REGION Network 34: 6. Авария - застрял ротаметр
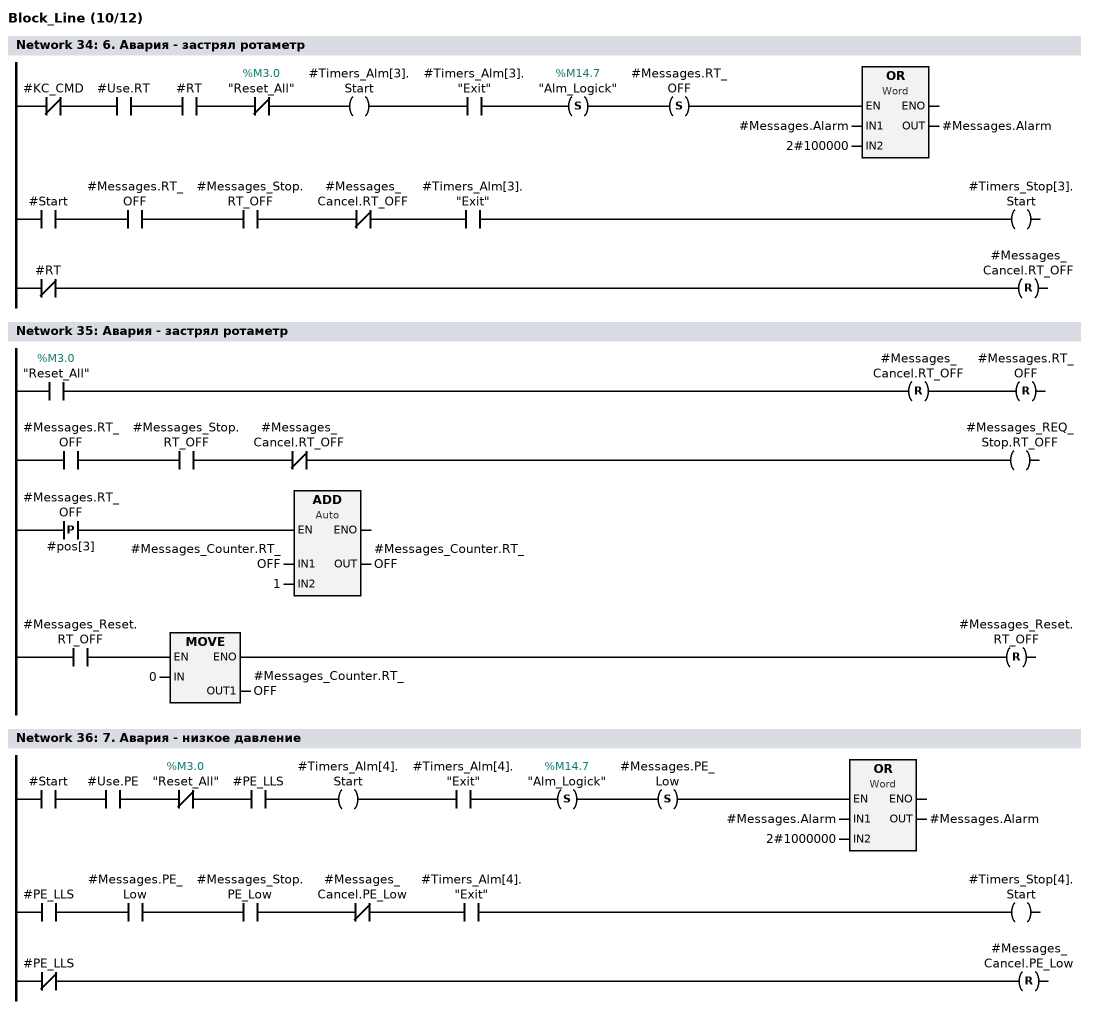
   #Timers_Alm[3].Start := NOT #KC_CMD AND #Use.RT AND #RT AND NOT "Reset_All";
   IF NOT #KC_CMD AND #Use.RT AND #RT AND NOT "Reset_All" AND #Timers_Alm[3]."Exit" THEN
       "Alm_Logick" := TRUE;
       #Messages.RT_OFF := TRUE;
       #Messages.Alarm := #Messages.Alarm OR 2#100000;
   END_IF;
   #Timers_Stop[3].Start := #Start AND #Messages.RT_OFF AND #Messages_Stop.RT_OFF AND NOT #Messages_Cancel.RT_OFF AND #Timers_Alm[3]."Exit";
   IF NOT #RT THEN #Messages_Cancel.RT_OFF := FALSE; END_IF;
END_REGION

REGION Network 35: Авария - застрял ротаметр
   RUNG wire#powerrail
      Contact( "Reset_All" )
      R_Coil( #Messages_Cancel.RT_OFF )
      R_Coil( #Messages.RT_OFF )
   END_RUNG
   RUNG wire#powerrail
      Contact( #Messages.RT_OFF )
      Contact( #Messages_Stop.RT_OFF )
      I_Contact( #Messages_Cancel.RT_OFF )
      Coil( #Messages_REQ_Stop.RT_OFF )
   END_RUNG
   RUNG wire#powerrail
      P_Contact(operand := #Messages.RT_OFF, bit := #pos[3])
      Add(in1 := #Messages_Counter.RT_OFF, in2 := 1, out => #Messages_Counter.RT_OFF)
   END_RUNG
   RUNG wire#powerrail
      Contact( #Messages_Reset.RT_OFF )
      Move(in := 0, out1 => #Messages_Counter.RT_OFF)
      R_Coil( #Messages_Reset.RT_OFF )
   END_RUNG
   // the same network as SCL:
   IF "Reset_All" THEN
       #Messages_Cancel.RT_OFF := FALSE;
       #Messages.RT_OFF := FALSE;
   END_IF;
   #Messages_REQ_Stop.RT_OFF := #Messages.RT_OFF AND #Messages_Stop.RT_OFF AND NOT #Messages_Cancel.RT_OFF;
   #_w1 := #Messages.RT_OFF AND NOT #pos[3];   // rising edge of #Messages.RT_OFF
   #pos[3] := #Messages.RT_OFF;
   IF #_w1 THEN #Messages_Counter.RT_OFF := #Messages_Counter.RT_OFF + 1; END_IF;
   IF #Messages_Reset.RT_OFF THEN
       #Messages_Counter.RT_OFF := 0;
       #Messages_Reset.RT_OFF := FALSE;
   END_IF;
END_REGION

REGION Network 36: 7. Авария - низкое давление
   #Timers_Alm[4].Start := #Start AND #Use.PE AND NOT "Reset_All" AND #PE_LLS;
   IF #Start AND #Use.PE AND NOT "Reset_All" AND #PE_LLS AND #Timers_Alm[4]."Exit" THEN
       "Alm_Logick" := TRUE;
       #Messages.PE_Low := TRUE;
       #Messages.Alarm := #Messages.Alarm OR 2#1000000;
   END_IF;
   #Timers_Stop[4].Start := #PE_LLS AND #Messages.PE_Low AND #Messages_Stop.PE_Low AND NOT #Messages_Cancel.PE_Low AND #Timers_Alm[4]."Exit";
   IF NOT #PE_LLS THEN #Messages_Cancel.PE_Low := FALSE; END_IF;
END_REGION

REGION Network 37: Авария - низкое давление
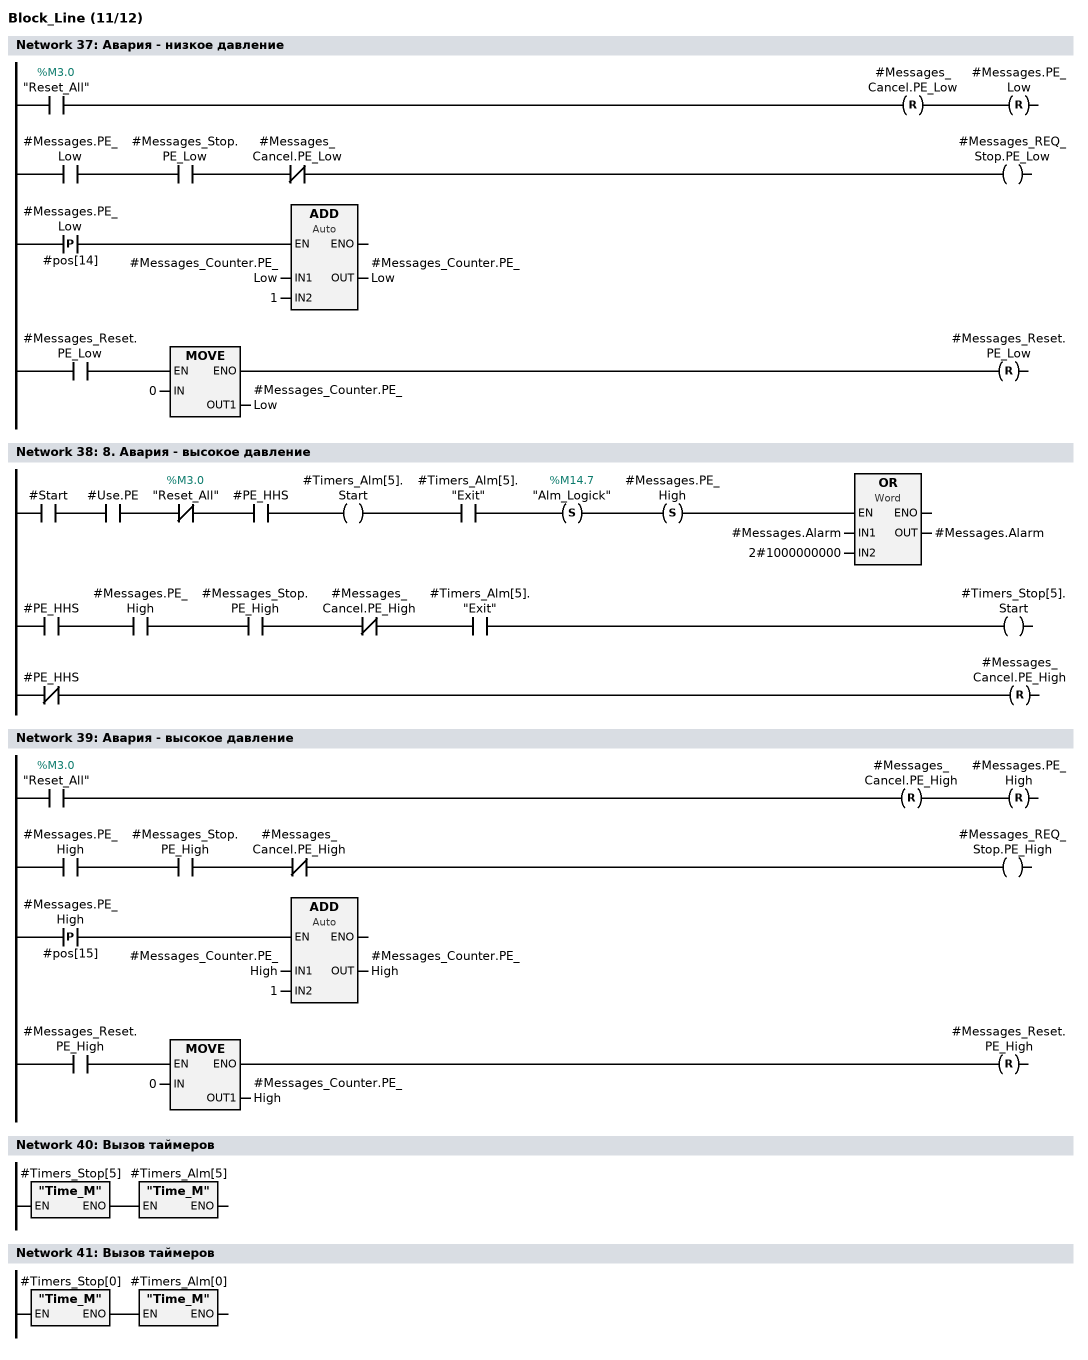
   RUNG wire#powerrail
      Contact( "Reset_All" )
      R_Coil( #Messages_Cancel.PE_Low )
      R_Coil( #Messages.PE_Low )
   END_RUNG
   RUNG wire#powerrail
      Contact( #Messages.PE_Low )
      Contact( #Messages_Stop.PE_Low )
      I_Contact( #Messages_Cancel.PE_Low )
      Coil( #Messages_REQ_Stop.PE_Low )
   END_RUNG
   RUNG wire#powerrail
      P_Contact(operand := #Messages.PE_Low, bit := #pos[14])
      Add(in1 := #Messages_Counter.PE_Low, in2 := 1, out => #Messages_Counter.PE_Low)
   END_RUNG
   RUNG wire#powerrail
      Contact( #Messages_Reset.PE_Low )
      Move(in := 0, out1 => #Messages_Counter.PE_Low)
      R_Coil( #Messages_Reset.PE_Low )
   END_RUNG
   // the same network as SCL:
   IF "Reset_All" THEN
       #Messages_Cancel.PE_Low := FALSE;
       #Messages.PE_Low := FALSE;
   END_IF;
   #Messages_REQ_Stop.PE_Low := #Messages.PE_Low AND #Messages_Stop.PE_Low AND NOT #Messages_Cancel.PE_Low;
   #_w1 := #Messages.PE_Low AND NOT #pos[14];   // rising edge of #Messages.PE_Low
   #pos[14] := #Messages.PE_Low;
   IF #_w1 THEN #Messages_Counter.PE_Low := #Messages_Counter.PE_Low + 1; END_IF;
   IF #Messages_Reset.PE_Low THEN
       #Messages_Counter.PE_Low := 0;
       #Messages_Reset.PE_Low := FALSE;
   END_IF;
END_REGION

REGION Network 38: 8. Авария - высокое давление
   #Timers_Alm[5].Start := #Start AND #Use.PE AND NOT "Reset_All" AND #PE_HHS;
   IF #Start AND #Use.PE AND NOT "Reset_All" AND #PE_HHS AND #Timers_Alm[5]."Exit" THEN
       "Alm_Logick" := TRUE;
       #Messages.PE_High := TRUE;
       #Messages.Alarm := #Messages.Alarm OR 2#1000000000;
   END_IF;
   #Timers_Stop[5].Start := #PE_HHS AND #Messages.PE_High AND #Messages_Stop.PE_High AND NOT #Messages_Cancel.PE_High AND #Timers_Alm[5]."Exit";
   IF NOT #PE_HHS THEN #Messages_Cancel.PE_High := FALSE; END_IF;
END_REGION

REGION Network 39: Авария - высокое давление
   RUNG wire#powerrail
      Contact( "Reset_All" )
      R_Coil( #Messages_Cancel.PE_High )
      R_Coil( #Messages.PE_High )
   END_RUNG
   RUNG wire#powerrail
      Contact( #Messages.PE_High )
      Contact( #Messages_Stop.PE_High )
      I_Contact( #Messages_Cancel.PE_High )
      Coil( #Messages_REQ_Stop.PE_High )
   END_RUNG
   RUNG wire#powerrail
      P_Contact(operand := #Messages.PE_High, bit := #pos[15])
      Add(in1 := #Messages_Counter.PE_High, in2 := 1, out => #Messages_Counter.PE_High)
   END_RUNG
   RUNG wire#powerrail
      Contact( #Messages_Reset.PE_High )
      Move(in := 0, out1 => #Messages_Counter.PE_High)
      R_Coil( #Messages_Reset.PE_High )
   END_RUNG
   // the same network as SCL:
   IF "Reset_All" THEN
       #Messages_Cancel.PE_High := FALSE;
       #Messages.PE_High := FALSE;
   END_IF;
   #Messages_REQ_Stop.PE_High := #Messages.PE_High AND #Messages_Stop.PE_High AND NOT #Messages_Cancel.PE_High;
   #_w1 := #Messages.PE_High AND NOT #pos[15];   // rising edge of #Messages.PE_High
   #pos[15] := #Messages.PE_High;
   IF #_w1 THEN #Messages_Counter.PE_High := #Messages_Counter.PE_High + 1; END_IF;
   IF #Messages_Reset.PE_High THEN
       #Messages_Counter.PE_High := 0;
       #Messages_Reset.PE_High := FALSE;
   END_IF;
END_REGION

REGION Network 40: Вызов таймеров
   RUNG wire#powerrail
      #Timers_Stop[5]()
      #Timers_Alm[5]()
   END_RUNG
   // the same network as SCL:
   #Timers_Stop[5](ENO => #_w1);   // "Time_M"
   IF #_w1 THEN
       #Timers_Alm[5]();   // "Time_M"
   END_IF;
END_REGION

REGION Network 41: Вызов таймеров
   RUNG wire#powerrail
      #Timers_Stop[0]()
      #Timers_Alm[0]()
   END_RUNG
   // the same network as SCL:
   #Timers_Stop[0](ENO => #_w1);   // "Time_M"
   IF #_w1 THEN
       #Timers_Alm[0]();   // "Time_M"
   END_IF;
END_REGION

REGION Network 42: Вызов таймеров
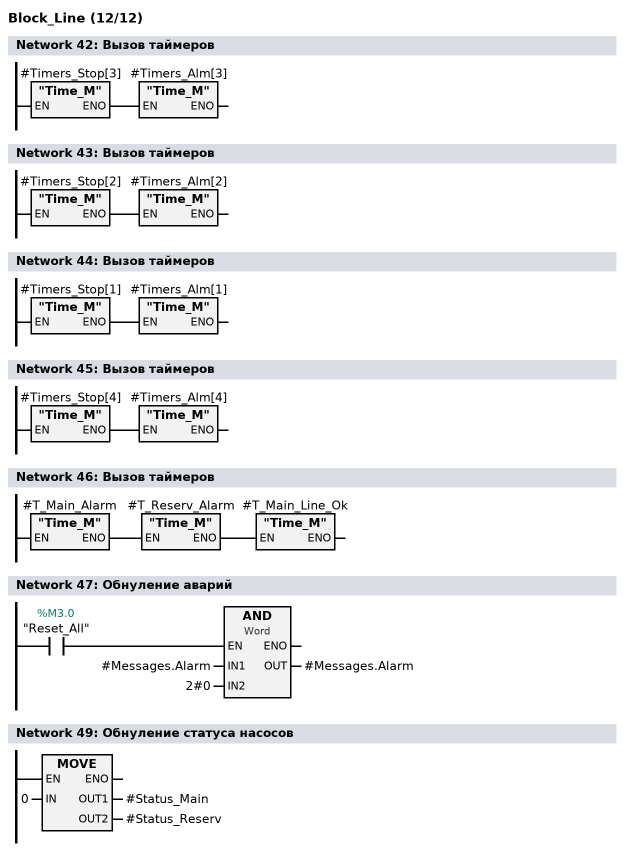
   RUNG wire#powerrail
      #Timers_Stop[3]()
      #Timers_Alm[3]()
   END_RUNG
   // the same network as SCL:
   #Timers_Stop[3](ENO => #_w1);   // "Time_M"
   IF #_w1 THEN
       #Timers_Alm[3]();   // "Time_M"
   END_IF;
END_REGION

REGION Network 43: Вызов таймеров
   RUNG wire#powerrail
      #Timers_Stop[2]()
      #Timers_Alm[2]()
   END_RUNG
   // the same network as SCL:
   #Timers_Stop[2](ENO => #_w1);   // "Time_M"
   IF #_w1 THEN
       #Timers_Alm[2]();   // "Time_M"
   END_IF;
END_REGION

REGION Network 44: Вызов таймеров
   RUNG wire#powerrail
      #Timers_Stop[1]()
      #Timers_Alm[1]()
   END_RUNG
   // the same network as SCL:
   #Timers_Stop[1](ENO => #_w1);   // "Time_M"
   IF #_w1 THEN
       #Timers_Alm[1]();   // "Time_M"
   END_IF;
END_REGION

REGION Network 45: Вызов таймеров
   RUNG wire#powerrail
      #Timers_Stop[4]()
      #Timers_Alm[4]()
   END_RUNG
   // the same network as SCL:
   #Timers_Stop[4](ENO => #_w1);   // "Time_M"
   IF #_w1 THEN
       #Timers_Alm[4]();   // "Time_M"
   END_IF;
END_REGION

REGION Network 46: Вызов таймеров
   RUNG wire#powerrail
      #T_Main_Alarm()
      #T_Reserv_Alarm()
      #T_Main_Line_Ok()
   END_RUNG
   // the same network as SCL:
   #T_Main_Alarm(ENO => #_w1);   // "Time_M"
   #T_Reserv_Alarm(EN := #_w1, ENO => #_w2);   // "Time_M"
   IF #_w2 THEN
       #T_Main_Line_Ok();   // "Time_M"
   END_IF;
END_REGION

REGION Network 47: Обнуление аварий
   RUNG wire#powerrail
      Contact( "Reset_All" )
      { S7_Templates := "SrcType := Word" } And(in1 := #Messages.Alarm, in2 := 2#0, out => #Messages.Alarm)
   END_RUNG
   // the same network as SCL:
   IF "Reset_All" THEN #Messages.Alarm := #Messages.Alarm AND 2#0; END_IF;
END_REGION

REGION Network 48: Обнуление Report
END_REGION

REGION Network 49: Обнуление статуса насосов
   RUNG wire#powerrail
      Move(in := 0, out1 => #Status_Main, out2 => #Status_Reserv)
   END_RUNG
   // the same network as SCL:
   #Status_Main := 0;
   #Status_Reserv := 0;
END_REGION
END_FUNCTION_BLOCK

FUNCTION_BLOCK "PID_ex"   // FB99, LAD
{ S7_Optimized_Access := 'FALSE' }
VERSION : 0.1
// stored: AutoNumber false, IsIECCheckEnabled false, SetENOAutomatically false, UDAEnableTagReadback false
   VAR_INPUT
      Start : Bool;
      SP_A : Real;   // Уставка
      Value : Real;   // Показания датчика
   END_VAR
   VAR_OUTPUT
      PWM : Bool;   // ШИМ-выход ПИД-регулятора
      Result : Real;   // Управляющее воздействие
   END_VAR
   VAR DB_SPECIFIC
      CMD { S7_SetPoint := 'True'} : "CMD";
      SP_M : Real;
      SP : Real;
      x { S7_SetPoint := 'True'} : Real := 1.0;   // Поправка уставки и датчика
      SP_x : Real;   // Домноженная уставка
      Value_x : Real;   // Домноженный датчик
      Buffer : Real;   // Промежуточное значение
      PID_Output : Real;   // Выход ПИД-регулятора
      PID_Hand : Real;   // Ручное задание выхода ПИД-регулятора
      Sys : Struct   // Системные параметры
         Err_Ack : Bool;   // Подтверждение аварии
         Alm_SP_H : Bool;   // Авария уставки - превышение
         Alm_SP_L : Bool;   // Авария уставки - занижение
         Alm_In_H : Bool;   // Авария датчика - превышение
         Alm_In_L : Bool;   // Авария датчика - занижение
         Activate : Bool;   // Активировать ПИД
         Error_code : DWord;   // Код аварии
         Warning_code : DWord;   // Код предупреждения
         "Type" : Int := 1;   // Режим работы
         State : Int;   // Состояние
         Mode : Int := 3;   // Режим
      END_STRUCT;
      Settings : Struct   // Рабочие параметры
         SP_P { S7_SetPoint := 'True'} : Real := 1.5;   // Коэффициент пропорциональности
         SP_Ti { S7_SetPoint := 'True'} : Real := 150.0;   // Время интегрирования
         SP_Td { S7_SetPoint := 'True'} : Real;   // Время дифференцирования
         SP_Cycle { S7_SetPoint := 'True'} : Real := 0.2;   // Время цикла
         Max_SP { S7_SetPoint := 'True'} : Real := 500.0;   // Максимальное значение уставки
         Min_SP { S7_SetPoint := 'True'} : Real := -500.0;   // Минимальное значение уставки
         Max_in { S7_SetPoint := 'True'} : Real := 500.0;   // Максимальное значение датчика
         Min_in { S7_SetPoint := 'True'} : Real := -500.0;   // Минимальное значение датчика
         Max_out { S7_SetPoint := 'True'} : Real := 100.0;   // Максимальное значение выхода
         Min_out { S7_SetPoint := 'True'} : Real := 0.0;   // Минимальное значение выхода
         DeadBand { S7_SetPoint := 'True'} : Real := 1.0;   // Мёртвая зона
         Max : Real;   // Верняя граница мёртвой зоны
         Min : Real;   // Нижняя граница мёртвой зоны
      END_STRUCT;
   END_VAR
   VAR
      PID { S7_SetPoint := 'True'} : PID_Compact;   // ПИД
      Converter : "Converter";   // Конвертер выхода
      Conveter_Back : "Converter";   // Конвертер Hand_SP в 0..100
      C { S7_SetPoint := 'True'} : "Time_R";   // Частота вызова ПИД на обработку
   END_VAR
   VAR DB_SPECIFIC
      pos : Array[0..15] of Bool;
   END_VAR
   VAR_TEMP
      x0 : Real;
   END_VAR
   // CMD.Start_A := true;
   // Converter.Max_In := 100.0;
   // Conveter_Back.Max_Out := 100.0;
   VAR_TEMP   // added for the SCL form of the ladder/FBD networks
      _w1 : Bool;
      _w2 : Bool;
   END_VAR
BEGIN

REGION Network 1: Сброс ПИД
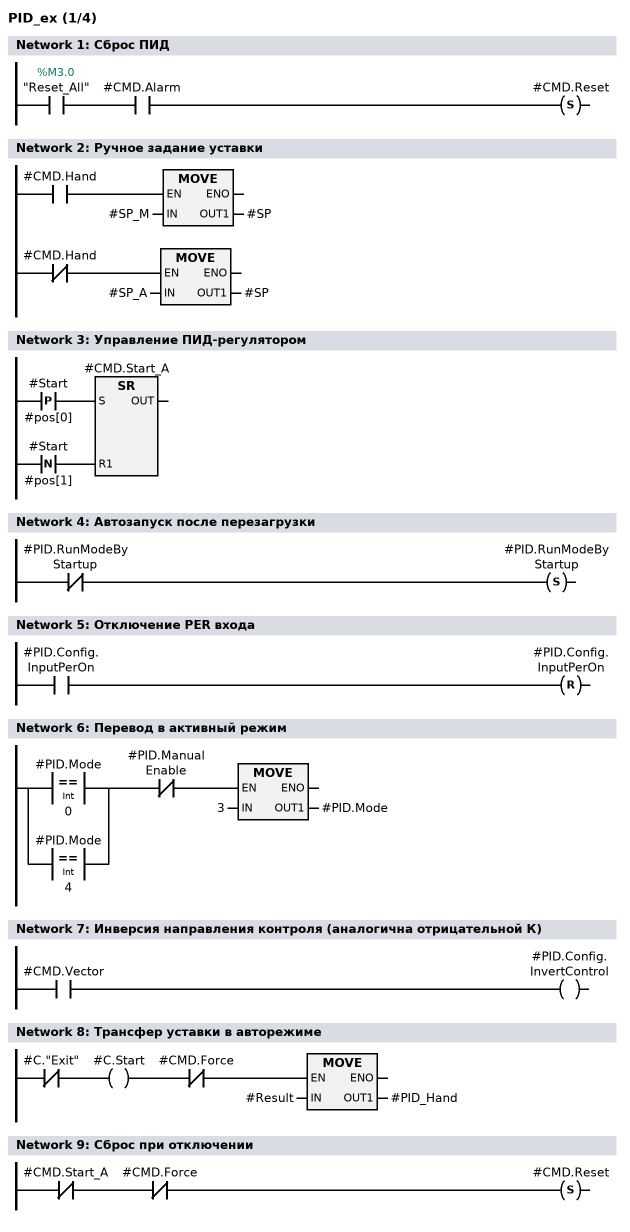
   RUNG wire#powerrail
      Contact( "Reset_All" )
      Contact( #CMD.Alarm )
      S_Coil( #CMD.Reset )
   END_RUNG
   // the same network as SCL:
   IF "Reset_All" AND #CMD.Alarm THEN #CMD.Reset := TRUE; END_IF;
END_REGION

REGION Network 2: Ручное задание уставки
   RUNG wire#powerrail
      Contact( #CMD.Hand )
      Move(in := #SP_M, out1 => #SP)
   END_RUNG
   RUNG wire#powerrail
      I_Contact( #CMD.Hand )
      Move(in := #SP_A, out1 => #SP)
   END_RUNG
   // the same network as SCL:
   IF #CMD.Hand THEN #SP := #SP_M; END_IF;
   IF NOT #CMD.Hand THEN #SP := #SP_A; END_IF;
END_REGION

REGION Network 3: Управление ПИД-регулятором
   RUNG wire#powerrail
      P_Contact(operand := #Start, bit := #pos[0])
      S_SR(operand := #CMD.Start_A, r1 := wire#w1)
   END_RUNG
   RUNG wire#powerrail
      N_Contact(operand := #Start, bit := #pos[1])
   END_RUNG wire#w1
   // the same network as SCL:
   #_w1 := #Start AND NOT #pos[0];   // rising edge of #Start
   #pos[0] := #Start;
   #_w2 := NOT #Start AND #pos[1];   // falling edge of #Start
   #pos[1] := #Start;
   IF #_w1 THEN
       #CMD.Start_A := TRUE;   // SR flip-flop
   END_IF;
   IF #_w2 THEN #CMD.Start_A := FALSE; END_IF;
END_REGION

REGION Network 4: Автозапуск после перезагрузки
   RUNG wire#powerrail
      I_Contact( #PID.RunModeByStartup )
      S_Coil( #PID.RunModeByStartup )
   END_RUNG
   // the same network as SCL:
   IF NOT #PID.RunModeByStartup THEN #PID.RunModeByStartup := TRUE; END_IF;
END_REGION

REGION Network 5: Отключение PER входа
   RUNG wire#powerrail
      Contact( #PID.Config.InputPerOn )
      R_Coil( #PID.Config.InputPerOn )
   END_RUNG
   // the same network as SCL:
   IF #PID.Config.InputPerOn THEN #PID.Config.InputPerOn := FALSE; END_IF;
END_REGION

REGION Network 6: Перевод в активный режим
   RUNG wire#powerrail
      { S7_Templates := "SrcType := Int" } EQ_Contact(in1 := #PID.Mode, in2 := 0)
      wire#w1
      I_Contact( #PID.ManualEnable )
      { S7_GenerateENO := "TRUE" } Move(in := 3, out1 => #PID.Mode)
   END_RUNG
   RUNG wire#powerrail
      { S7_Templates := "SrcType := Int" } EQ_Contact(in1 := #PID.Mode, in2 := 4)
   END_RUNG wire#w1
   // the same network as SCL:
   IF ((#PID.Mode = 0) OR (#PID.Mode = 4)) AND NOT #PID.ManualEnable THEN #PID.Mode := 3; END_IF;
END_REGION

REGION Network 7: Инверсия направления контроля (аналогична отрицательной К)
   RUNG wire#powerrail
      Contact( #CMD.Vector )
      Coil( #PID.Config.InvertControl )
   END_RUNG
   // the same network as SCL:
   #PID.Config.InvertControl := #CMD.Vector;
END_REGION

REGION Network 8: Трансфер уставки в авторежиме
   RUNG wire#powerrail
      I_Contact( #C."Exit" )
      Coil( #C.Start )
      I_Contact( #CMD.Force )
      Move(in := #Result, out1 => #PID_Hand)
   END_RUNG
   // the same network as SCL:
   #C.Start := NOT #C."Exit";
   IF NOT #C."Exit" AND NOT #CMD.Force THEN #PID_Hand := #Result; END_IF;
END_REGION

REGION Network 9: Сброс при отключении
   RUNG wire#powerrail
      I_Contact( #CMD.Start_A )
      I_Contact( #CMD.Force )
      S_Coil( #CMD.Reset )
   END_RUNG
   // the same network as SCL:
   IF NOT #CMD.Start_A AND NOT #CMD.Force THEN #CMD.Reset := TRUE; END_IF;
END_REGION

REGION Network 10: Активация после смены режима
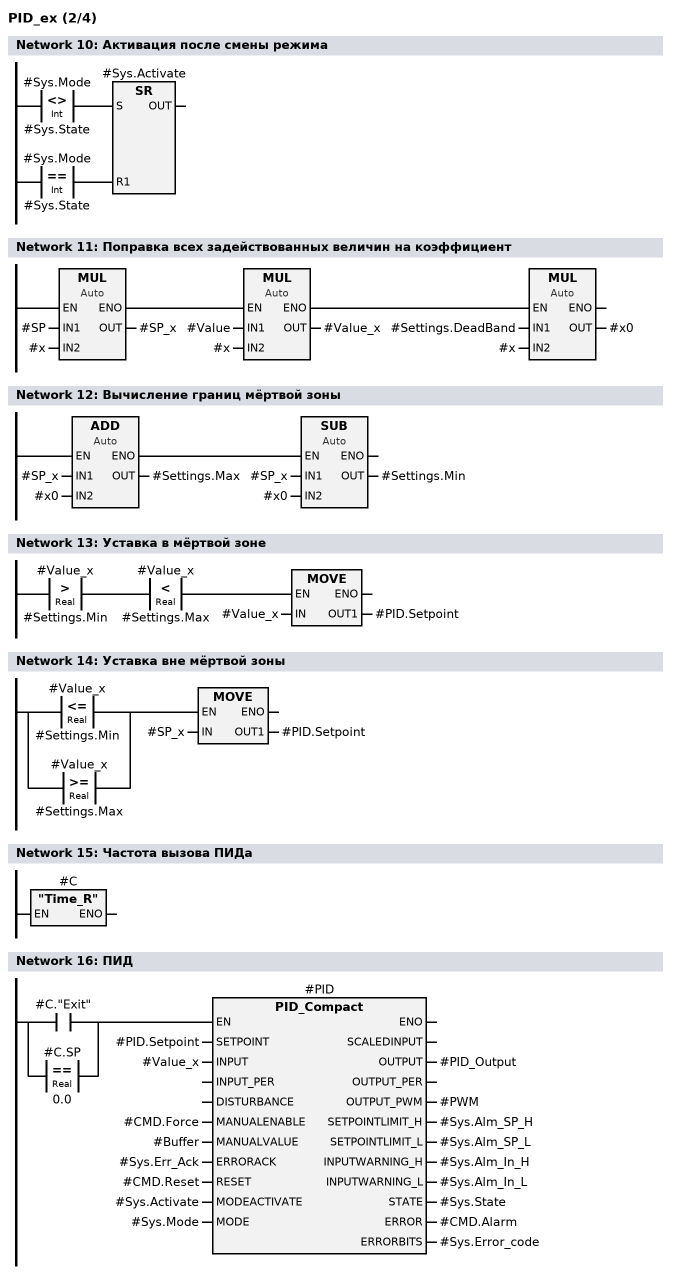
   RUNG wire#powerrail
      { S7_Templates := "SrcType := Int" } NE_Contact(in1 := #Sys.Mode, in2 := #Sys.State)
      S_SR(operand := #Sys.Activate, r1 := wire#w1)
   END_RUNG
   RUNG wire#powerrail
      { S7_Templates := "SrcType := Int" } EQ_Contact(in1 := #Sys.Mode, in2 := #Sys.State)
   END_RUNG wire#w1
   // the same network as SCL:
   IF #Sys.Mode <> #Sys.State THEN
       #Sys.Activate := TRUE;   // SR flip-flop
   END_IF;
   IF #Sys.Mode = #Sys.State THEN #Sys.Activate := FALSE; END_IF;
END_REGION

REGION Network 11: Поправка всех задействованных величин на коэффициент
   RUNG wire#powerrail
      Mul(in1 := #SP, in2 := #x, out => #SP_x)
      Mul(in1 := #Value, in2 := #x, out => #Value_x)
      Mul(in1 := #Settings.DeadBand, in2 := #x, out => #x0)
   END_RUNG
   // the same network as SCL:
   #SP_x := #SP * #x;
   #Value_x := #Value * #x;
   #x0 := #Settings.DeadBand * #x;
END_REGION

REGION Network 12: Вычисление границ мёртвой зоны
   RUNG wire#powerrail
      Add(in1 := #SP_x, in2 := #x0, out => #Settings.Max)
      Sub(in1 := #SP_x, in2 := #x0, out => #Settings.Min)
   END_RUNG
   // the same network as SCL:
   #Settings.Max := #SP_x + #x0;
   #Settings.Min := #SP_x - #x0;
END_REGION

REGION Network 13: Уставка в мёртвой зоне
   RUNG wire#powerrail
      { S7_Templates := "SrcType := Real" } GT_Contact(in1 := #Value_x, in2 := #Settings.Min)
      { S7_Templates := "SrcType := Real" } LT_Contact(in1 := #Value_x, in2 := #Settings.Max)
      Move(in := #Value_x, out1 => #PID.Setpoint)
   END_RUNG
   // the same network as SCL:
   IF (#Value_x > #Settings.Min) AND (#Value_x < #Settings.Max) THEN #PID.Setpoint := #Value_x; END_IF;
END_REGION

REGION Network 14: Уставка вне мёртвой зоны
   RUNG wire#powerrail
      { S7_Templates := "SrcType := Real" } LE_Contact(in1 := #Value_x, in2 := #Settings.Min)
      wire#w1
      Move(in := #SP_x, out1 => #PID.Setpoint)
   END_RUNG
   RUNG wire#powerrail
      { S7_Templates := "SrcType := Real" } GE_Contact(in1 := #Value_x, in2 := #Settings.Max)
   END_RUNG wire#w1
   // the same network as SCL:
   IF (#Value_x <= #Settings.Min) OR (#Value_x >= #Settings.Max) THEN #PID.Setpoint := #SP_x; END_IF;
END_REGION

REGION Network 15: Частота вызова ПИДа
   RUNG wire#powerrail
      #C()
   END_RUNG
   // the same network as SCL:
   #C();   // "Time_R"
END_REGION

REGION Network 16: ПИД
   RUNG wire#powerrail
      Contact( #C."Exit" )
      wire#w1
      #PID.PID_Compact(Setpoint := #PID.Setpoint, Input := #Value_x, Input_PER :=, Disturbance :=, ManualEnable := #CMD.Force, ManualValue := #Buffer, ErrorAck := #Sys.Err_Ack, Reset := #CMD.Reset, ModeActivate := #Sys.Activate, Mode := #Sys.Mode, ScaledInput =>, Output => #PID_Output, Output_PER =>, Output_PWM => #PWM, SetpointLimit_H => #Sys.Alm_SP_H, SetpointLimit_L => #Sys.Alm_SP_L, InputWarning_H => #Sys.Alm_In_H, InputWarning_L => #Sys.Alm_In_L, State => #Sys.State, Error => #CMD.Alarm, ErrorBits => #Sys.Error_code)
   END_RUNG
   RUNG wire#powerrail
      { S7_Templates := "SrcType := Real" } EQ_Contact(in1 := #C.SP, in2 := 0.0)
   END_RUNG wire#w1
   // the same network as SCL:
   IF #C."Exit" OR (#C.SP = 0.0) THEN
       #PID(Setpoint := #PID.Setpoint,   // PID_Compact
            Input := #Value_x,
            ManualEnable := #CMD.Force,
            ManualValue := #Buffer,
            ErrorAck := #Sys.Err_Ack,
            Reset := #CMD.Reset,
            ModeActivate := #Sys.Activate,
            Mode := #Sys.Mode,
            Output => #PID_Output,
            Output_PWM => #PWM,
            SetpointLimit_H => #Sys.Alm_SP_H,
            SetpointLimit_L => #Sys.Alm_SP_L,
            InputWarning_H => #Sys.Alm_In_H,
            InputWarning_L => #Sys.Alm_In_L,
            State => #Sys.State,
            Error => #CMD.Alarm,
            ErrorBits => #Sys.Error_code);
   END_IF;
END_REGION

REGION Network 17: Обратное масштабирование в ручном режиме
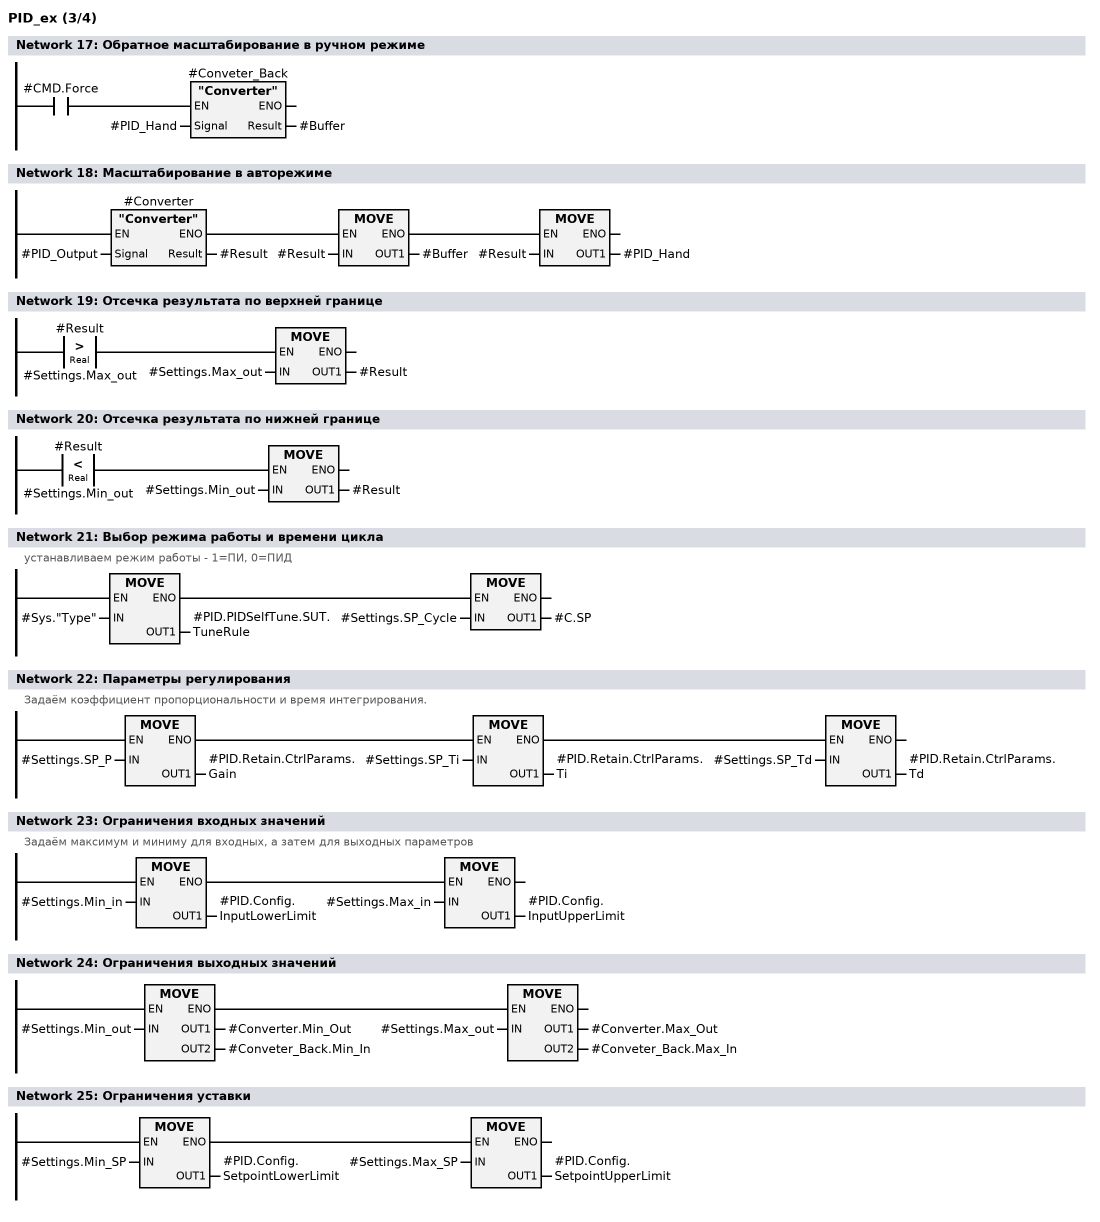
   RUNG wire#powerrail
      Contact( #CMD.Force )
      #Conveter_Back(Signal := #PID_Hand, Result => #Buffer)
   END_RUNG
   // the same network as SCL:
   IF #CMD.Force THEN
       #Conveter_Back(Signal := #PID_Hand, Result => #Buffer);   // "Converter"
   END_IF;
END_REGION

REGION Network 18: Масштабирование в авторежиме
   RUNG wire#powerrail
      #Converter(Signal := #PID_Output, Result => #Result)
      { S7_GenerateENO := "TRUE" } Move(in := #Result, out1 => #Buffer)
      { S7_GenerateENO := "TRUE" } Move(in := #Result, out1 => #PID_Hand)
   END_RUNG
   // the same network as SCL:
   // ENO of a box is taken as its EN; it also drops when the box reports an error
   #Converter(Signal := #PID_Output, Result => #Result, ENO => #_w1);   // "Converter"
   IF #_w1 THEN
       #Buffer := #Result;
       #PID_Hand := #Result;
   END_IF;
END_REGION

REGION Network 19: Отсечка результата по верхней границе
   RUNG wire#powerrail
      { S7_Templates := "SrcType := Real" } GT_Contact(in1 := #Result, in2 := #Settings.Max_out)
      Move(in := #Settings.Max_out, out1 => #Result)
   END_RUNG
   // the same network as SCL:
   IF #Result > #Settings.Max_out THEN #Result := #Settings.Max_out; END_IF;
END_REGION

REGION Network 20: Отсечка результата по нижней границе
   RUNG wire#powerrail
      { S7_Templates := "SrcType := Real" } LT_Contact(in1 := #Result, in2 := #Settings.Min_out)
      Move(in := #Settings.Min_out, out1 => #Result)
   END_RUNG
   // the same network as SCL:
   IF #Result < #Settings.Min_out THEN #Result := #Settings.Min_out; END_IF;
END_REGION

REGION Network 21: Выбор режима работы и времени цикла
   // устанавливаем режим работы - 1=ПИ, 0=ПИД
   RUNG wire#powerrail
      { S7_GenerateENO := "TRUE" } Move(in := #Sys."Type", out1 => #PID.PIDSelfTune.SUT.TuneRule)
      { S7_GenerateENO := "TRUE" } Move(in := #Settings.SP_Cycle, out1 => #C.SP)
   END_RUNG
   // the same network as SCL:
   // ENO of a box is taken as its EN; it also drops when the box reports an error
   #PID.PIDSelfTune.SUT.TuneRule := #Sys."Type";
   #C.SP := #Settings.SP_Cycle;
END_REGION

REGION Network 22: Параметры регулирования
   // Задаём коэффициент пропорциональности и время интегрирования.
   RUNG wire#powerrail
      { S7_GenerateENO := "TRUE" } Move(in := #Settings.SP_P, out1 => #PID.Retain.CtrlParams.Gain)
      { S7_GenerateENO := "TRUE" } Move(in := #Settings.SP_Ti, out1 => #PID.Retain.CtrlParams.Ti)
      { S7_GenerateENO := "TRUE" } Move(in := #Settings.SP_Td, out1 => #PID.Retain.CtrlParams.Td)
   END_RUNG
   // the same network as SCL:
   // ENO of a box is taken as its EN; it also drops when the box reports an error
   #PID.Retain.CtrlParams.Gain := #Settings.SP_P;
   #PID.Retain.CtrlParams.Ti := #Settings.SP_Ti;
   #PID.Retain.CtrlParams.Td := #Settings.SP_Td;
END_REGION

REGION Network 23: Ограничения входных значений
   // Задаём максимум и миниму для входных, а затем для выходных параметров
   RUNG wire#powerrail
      { S7_GenerateENO := "TRUE" } Move(in := #Settings.Min_in, out1 => #PID.Config.InputLowerLimit)
      { S7_GenerateENO := "TRUE" } Move(in := #Settings.Max_in, out1 => #PID.Config.InputUpperLimit)
   END_RUNG
   // the same network as SCL:
   // ENO of a box is taken as its EN; it also drops when the box reports an error
   #PID.Config.InputLowerLimit := #Settings.Min_in;
   #PID.Config.InputUpperLimit := #Settings.Max_in;
END_REGION

REGION Network 24: Ограничения выходных значений
   RUNG wire#powerrail
      { S7_GenerateENO := "TRUE" } Move(in := #Settings.Min_out, out1 => #Converter.Min_Out, out2 => #Conveter_Back.Min_In)
      { S7_GenerateENO := "TRUE" } Move(in := #Settings.Max_out, out1 => #Converter.Max_Out, out2 => #Conveter_Back.Max_In)
   END_RUNG
   // the same network as SCL:
   // ENO of a box is taken as its EN; it also drops when the box reports an error
   #Converter.Min_Out := #Settings.Min_out;
   #Conveter_Back.Min_In := #Settings.Min_out;
   #Converter.Max_Out := #Settings.Max_out;
   #Conveter_Back.Max_In := #Settings.Max_out;
END_REGION

REGION Network 25: Ограничения уставки
   RUNG wire#powerrail
      { S7_GenerateENO := "TRUE" } Move(in := #Settings.Min_SP, out1 => #PID.Config.SetpointLowerLimit)
      { S7_GenerateENO := "TRUE" } Move(in := #Settings.Max_SP, out1 => #PID.Config.SetpointUpperLimit)
   END_RUNG
   // the same network as SCL:
   // ENO of a box is taken as its EN; it also drops when the box reports an error
   #PID.Config.SetpointLowerLimit := #Settings.Min_SP;
   #PID.Config.SetpointUpperLimit := #Settings.Max_SP;
END_REGION

REGION Network 26: Сброс сброса
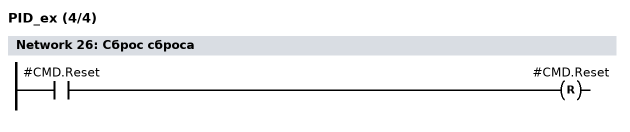
   RUNG wire#powerrail
      Contact( #CMD.Reset )
      R_Coil( #CMD.Reset )
   END_RUNG
   // the same network as SCL:
   IF #CMD.Reset THEN #CMD.Reset := FALSE; END_IF;
END_REGION
END_FUNCTION_BLOCK

FUNCTION_BLOCK "DRV_Flow_old"   // FB115, LAD
{ S7_Optimized_Access := 'TRUE' }
VERSION : 0.1
// stored: AutoNumber false, IsIECCheckEnabled false, IsRetainMemResEnabled false, MemoryReserve 100, SetENOAutomatically false, UDAEnableTagReadback false
   VAR_INPUT
      Start : Bool;   // Старт
      Value : Real;   // Значение
   END_VAR
   VAR RETAIN
      Mode { S7_SetPoint := 'True'} : Bool;   // 0 - импульсный, 1 - аналоговый
   END_VAR
   VAR
      Lock : Bool;   // Блокировка учёта расхода воды
      pulse : Bool;   // Пульс
      Reset_All : Bool;   // Сброс общего счётчика
      Reset_Now : Bool;   // Сброс суточного счётчика
      Reset_Last : Bool;   // Сброс последнего счётчика
      Reset_Seans : Bool;   // Сброс счёта за сеанс
      Reset_Any : Bool;   // Сброс произвольного измерения
      Save : Bool;   // Сохранить данные за сеанс
      SaveDay : Bool;   // Сохранить данные за сутки
   END_VAR
   VAR RETAIN
      Fast_Mode { S7_SetPoint := 'True'} : Bool := True;   // Режим частых импульсов
   END_VAR
   VAR
      Inverse : Bool;   // Инверсия
      pos : Array[0..7] of Bool;   // Вспомогательные переменные
      clock { S7_SetPoint := 'True'} : Real := 0.01;   // Контроль связи 1 Гц
   END_VAR
   VAR RETAIN
      Weight { S7_SetPoint := 'True'} : Real := 1.0;   // Вес импульса
   END_VAR
   VAR
      Weight_S : Real;   // Расход за секунду
   END_VAR
   VAR RETAIN
      All { S7_SetPoint := 'True'} : Real;   // Полный расход
      Any { S7_SetPoint := 'True'} : Real;   // Произвольное измерение
      Seans { S7_SetPoint := 'True'} : Real;   // Расход за сеанс работы
      Seans_Last { S7_SetPoint := 'True'} : Real;   // Расход за прошлый сеанс
      Flow_Today { S7_SetPoint := 'True'} : Real;   // Расход за текущее измерение
      Flow_LastDay { S7_SetPoint := 'True'} : Real;   // Расход за прошлое измерение
      Flow_Lock_All { S7_SetPoint := 'True'} : Real;   // Неучтённый расход
      Flow_Lock_Now { S7_SetPoint := 'True'} : Real;   // Текущий неучтенный расхрд
   END_VAR
   VAR
      Flow_S : Real;   // Расход в секунду по импульсам
      Flow_Speed : Real;   // Скорость потока л/ч
      Pulse_CNT : Real;   // Число импульсов за время измерения
      Flow_DTM : Real;   // Низкая скорость - проток в минуту
      Flow_DT : Real;   // Время между импульсами
      Flow_clock : Real;   // Не используется
      TimeControl : "Time_R";   // Время измерения
   END_VAR
   VAR RETAIN
      Day : Int;   // Текущая дата
      ADDR_Byte { S7_SetPoint := 'True'} : Int;   // Адрес входа на контроллере (Байт)
      ADDR_Bit { S7_SetPoint := 'True'} : Int;   // Адрес входа на контроллере (Бит)
   END_VAR
   VAR
      Filter { S7_SetPoint := 'True'} : "Filter";
      Time_DTL : DTL;
   END_VAR
   VAR_TEMP
      imp : Bool;
      start_x : Bool;
      m3 : Real;
   END_VAR
   VAR CONSTANT
      Minutes : Real := 60.0;
      Hour : Real := 3600.0;
   END_VAR
   // Filter.max := 100;
   VAR_TEMP   // added for the SCL form of the ladder/FBD networks
      _w1 : Bool;
      _w2 : Bool;
   END_VAR
BEGIN

REGION Network 1: Чтение сигнала
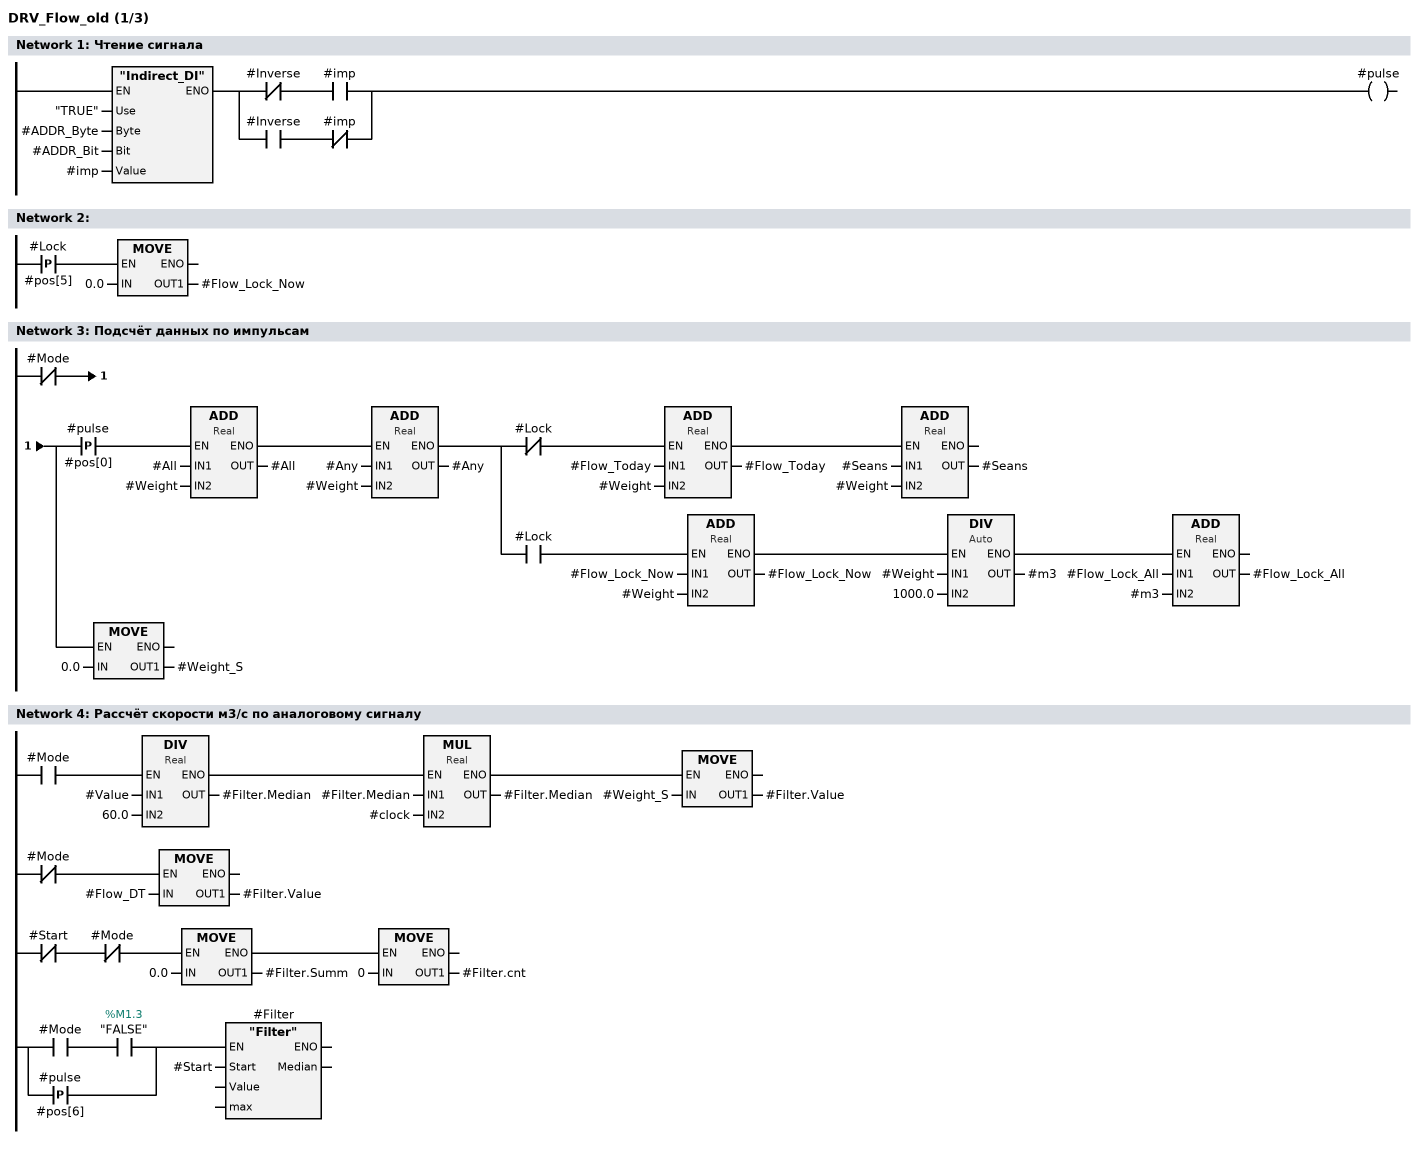
   RUNG wire#powerrail
      "Indirect_DI"(Use := "TRUE", "Byte" := #ADDR_Byte, Bit := #ADDR_Bit, Value := #imp)
      wire#w1
      I_Contact( #Inverse )
      Contact( #imp )
      wire#w2
      Coil( #pulse )
   END_RUNG
   RUNG wire#w1
      Contact( #Inverse )
      I_Contact( #imp )
   END_RUNG wire#w2
   // the same network as SCL:
   "Indirect_DI"(Use := "TRUE", "Byte" := #ADDR_Byte, Bit := #ADDR_Bit, Value := #imp, ENO => #_w1);
   #pulse := #_w1 AND ((NOT #Inverse AND #imp) OR (#Inverse AND NOT #imp));
END_REGION

REGION Network 2
   RUNG wire#powerrail
      P_Contact(operand := #Lock, bit := #pos[5])
      Move(in := 0.0, out1 => #Flow_Lock_Now)
   END_RUNG
   // the same network as SCL:
   #_w1 := #Lock AND NOT #pos[5];   // rising edge of #Lock
   #pos[5] := #Lock;
   IF #_w1 THEN #Flow_Lock_Now := 0.0; END_IF;
END_REGION

REGION Network 3: Подсчёт данных по импульсам
   RUNG wire#powerrail
      I_Contact( #Mode )
      wire#w1
      P_Contact(operand := #pulse, bit := #pos[0])
      { S7_Templates := "SrcType := Real"; S7_GenerateENO := "TRUE" } Add(in1 := #All, in2 := #Weight, out => #All)
      { S7_Templates := "SrcType := Real"; S7_GenerateENO := "TRUE" } Add(in1 := #Any, in2 := #Weight, out => #Any)
      wire#w2
      I_Contact( #Lock )
      { S7_Templates := "SrcType := Real"; S7_GenerateENO := "TRUE" } Add(in1 := #Flow_Today, in2 := #Weight, out => #Flow_Today)
      { S7_Templates := "SrcType := Real"; S7_GenerateENO := "TRUE" } Add(in1 := #Seans, in2 := #Weight, out => #Seans)
   END_RUNG
   RUNG wire#w2
      Contact( #Lock )
      { S7_Templates := "SrcType := Real"; S7_GenerateENO := "TRUE" } Add(in1 := #Flow_Lock_Now, in2 := #Weight, out => #Flow_Lock_Now)
      Div(in1 := #Weight, in2 := 1000.0, out => #m3)
      { S7_Templates := "SrcType := Real"; S7_GenerateENO := "TRUE" } Add(in1 := #Flow_Lock_All, in2 := #m3, out => #Flow_Lock_All)
   END_RUNG
   RUNG wire#w1
      Move(in := 0.0, out1 => #Weight_S)
   END_RUNG
   // the same network as SCL:
   // ENO of a box is taken as its EN; it also drops when the box reports an error
   #_w1 := NOT #Mode AND #pulse AND NOT #pos[0];   // rising edge of #pulse
   #pos[0] := #pulse;
   IF #_w1 THEN
       #All := #All + #Weight;
       #Any := #Any + #Weight;
   END_IF;
   IF #_w1 AND NOT #Lock THEN
       #Flow_Today := #Flow_Today + #Weight;
       #Seans := #Seans + #Weight;
   END_IF;
   IF #_w1 AND #Lock THEN
       #Flow_Lock_Now := #Flow_Lock_Now + #Weight;
       #m3 := #Weight / 1000.0;
       #Flow_Lock_All := #Flow_Lock_All + #m3;
   END_IF;
   IF NOT #Mode THEN #Weight_S := 0.0; END_IF;
END_REGION

REGION Network 4: Рассчёт скорости м3/с по аналоговому сигналу
   RUNG wire#powerrail
      Contact( #Mode )
      { S7_Templates := "SrcType := Real"; S7_GenerateENO := "TRUE" } Div(in1 := #Value, in2 := 60.0, out => #Filter.Median)
      { S7_Templates := "SrcType := Real"; S7_GenerateENO := "TRUE" } Mul(in1 := #Filter.Median, in2 := #clock, out => #Filter.Median)
      Move(in := #Weight_S, out1 => #Filter.Value)
   END_RUNG
   RUNG wire#powerrail
      I_Contact( #Mode )
      Move(in := #Flow_DT, out1 => #Filter.Value)
   END_RUNG
   RUNG wire#powerrail
      I_Contact( #Start )
      I_Contact( #Mode )
      Move(in := 0.0, out1 => #Filter.Summ)
      Move(in := 0, out1 => #Filter.cnt)
   END_RUNG
   RUNG wire#powerrail
      Contact( #Mode )
      Contact( "FALSE" )
      wire#w1
      #Filter(Start := #Start, Value :=, max :=, Median =>)
   END_RUNG
   RUNG wire#powerrail
      P_Contact(operand := #pulse, bit := #pos[6])
   END_RUNG wire#w1
   // the same network as SCL:
   // ENO of a box is taken as its EN; it also drops when the box reports an error
   IF #Mode THEN
       #Filter.Median := #Value / 60.0;
       #Filter.Median := #Filter.Median * #clock;
       #Filter.Value := #Weight_S;
   END_IF;
   IF NOT #Mode THEN #Filter.Value := #Flow_DT; END_IF;
   IF NOT #Start AND NOT #Mode THEN
       #Filter.Summ := 0.0;
       #Filter.cnt := 0;
   END_IF;
   #_w1 := #pulse AND NOT #pos[6];   // rising edge of #pulse
   #pos[6] := #pulse;
   IF (#Mode AND "FALSE") OR #_w1 THEN
       #Filter(Start := #Start);   // "Filter"
   END_IF;
END_REGION

REGION Network 5: Подсчёт расхода по аналоговому сигналу
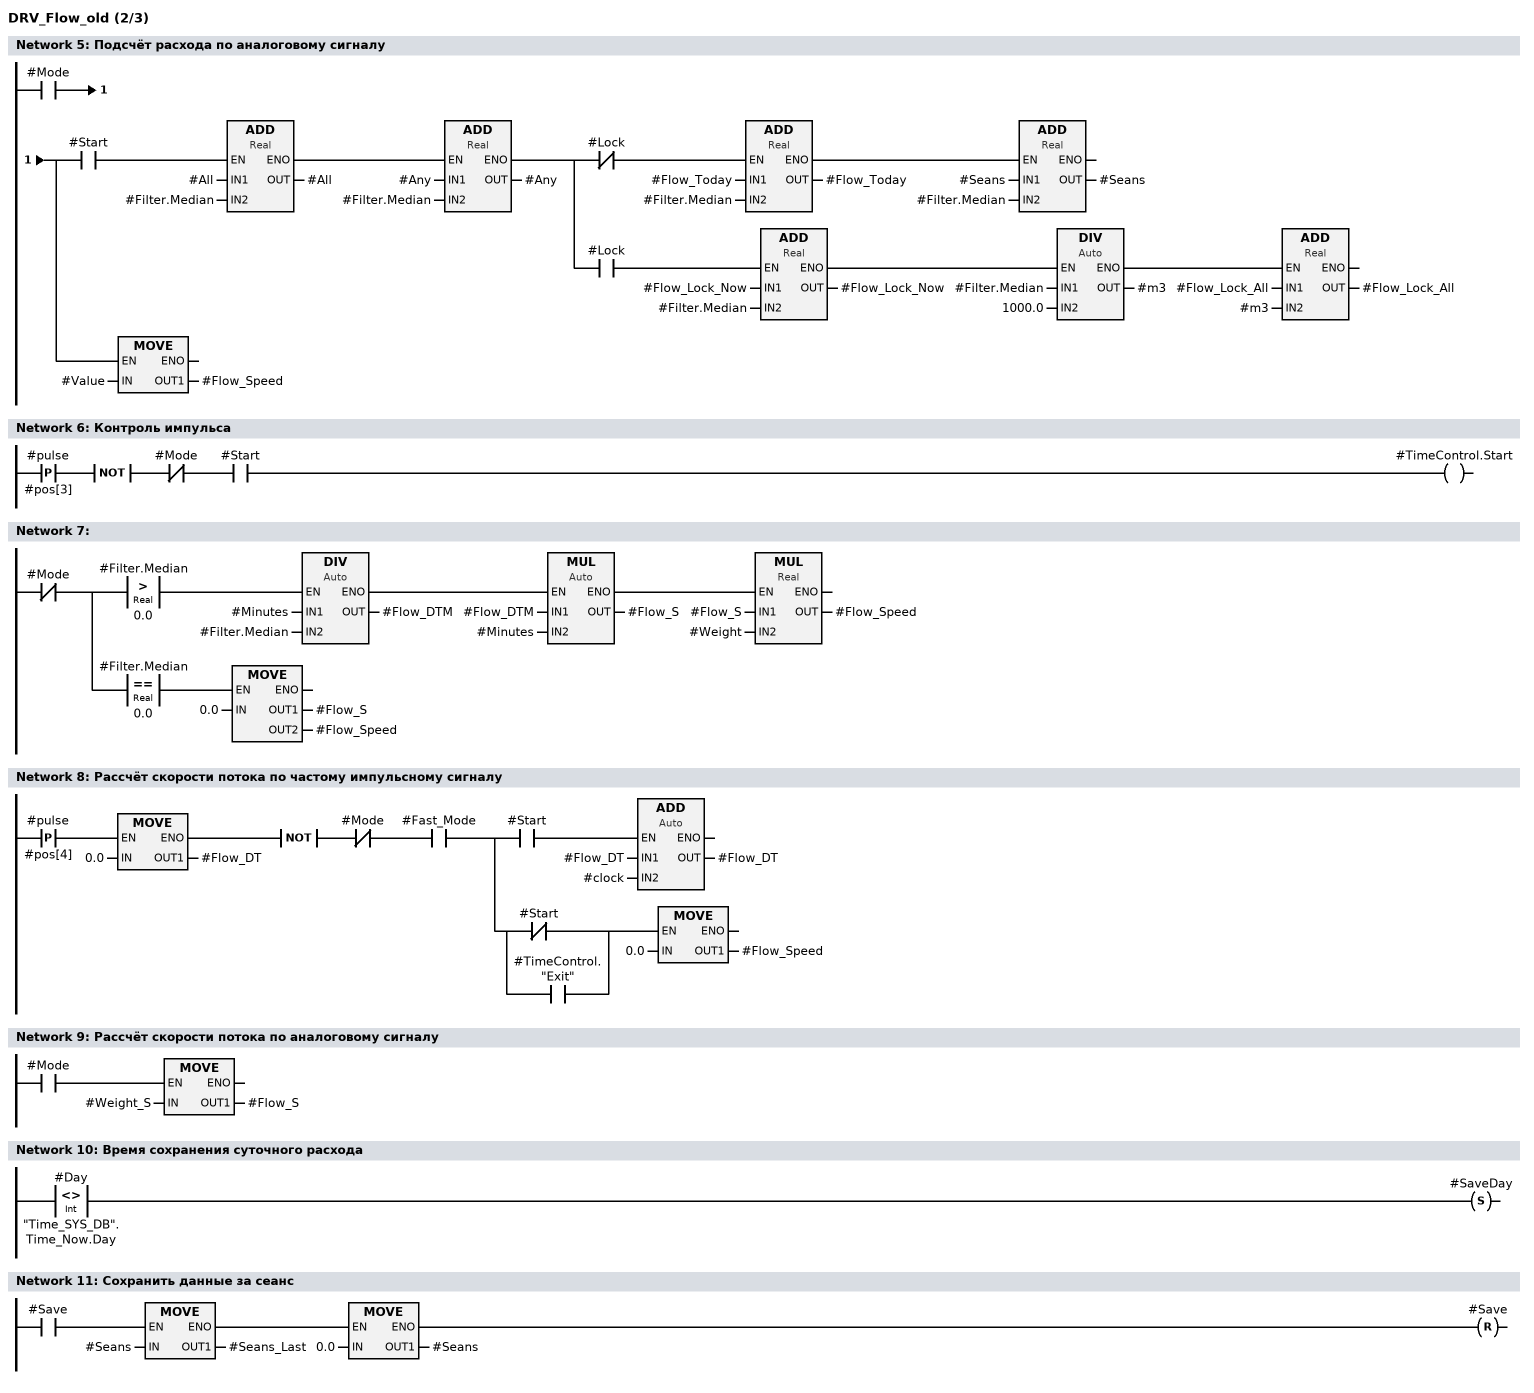
   RUNG wire#powerrail
      Contact( #Mode )
      wire#w1
      Contact( #Start )
      { S7_Templates := "SrcType := Real"; S7_GenerateENO := "TRUE" } Add(in1 := #All, in2 := #Filter.Median, out => #All)
      { S7_Templates := "SrcType := Real"; S7_GenerateENO := "TRUE" } Add(in1 := #Any, in2 := #Filter.Median, out => #Any)
      wire#w2
      I_Contact( #Lock )
      { S7_Templates := "SrcType := Real"; S7_GenerateENO := "TRUE" } Add(in1 := #Flow_Today, in2 := #Filter.Median, out => #Flow_Today)
      { S7_Templates := "SrcType := Real"; S7_GenerateENO := "TRUE" } Add(in1 := #Seans, in2 := #Filter.Median, out => #Seans)
   END_RUNG
   RUNG wire#w2
      Contact( #Lock )
      { S7_Templates := "SrcType := Real"; S7_GenerateENO := "TRUE" } Add(in1 := #Flow_Lock_Now, in2 := #Filter.Median, out => #Flow_Lock_Now)
      Div(in1 := #Filter.Median, in2 := 1000.0, out => #m3)
      { S7_Templates := "SrcType := Real"; S7_GenerateENO := "TRUE" } Add(in1 := #Flow_Lock_All, in2 := #m3, out => #Flow_Lock_All)
   END_RUNG
   RUNG wire#w1
      Move(in := #Value, out1 => #Flow_Speed)
   END_RUNG
   // the same network as SCL:
   // ENO of a box is taken as its EN; it also drops when the box reports an error
   #_w1 := #Mode AND #Start;
   IF #_w1 THEN
       #All := #All + #Filter.Median;
       #Any := #Any + #Filter.Median;
   END_IF;
   IF #_w1 AND NOT #Lock THEN
       #Flow_Today := #Flow_Today + #Filter.Median;
       #Seans := #Seans + #Filter.Median;
   END_IF;
   IF #_w1 AND #Lock THEN
       #Flow_Lock_Now := #Flow_Lock_Now + #Filter.Median;
       #m3 := #Filter.Median / 1000.0;
       #Flow_Lock_All := #Flow_Lock_All + #m3;
   END_IF;
   IF #Mode THEN #Flow_Speed := #Value; END_IF;
END_REGION

REGION Network 6: Контроль импульса
   RUNG wire#powerrail
      P_Contact(operand := #pulse, bit := #pos[3])
      Not()
      I_Contact( #Mode )
      Contact( #Start )
      Coil( #TimeControl.Start )
   END_RUNG
   // the same network as SCL:
   #_w1 := #pulse AND NOT #pos[3];   // rising edge of #pulse
   #pos[3] := #pulse;
   #TimeControl.Start := NOT #_w1 AND NOT #Mode AND #Start;
END_REGION

REGION Network 7
   RUNG wire#powerrail
      I_Contact( #Mode )
      wire#w1
      { S7_Templates := "SrcType := Real" } GT_Contact(in1 := #Filter.Median, in2 := 0.0)
      Div(in1 := #Minutes, in2 := #Filter.Median, out => #Flow_DTM)
      Mul(in1 := #Flow_DTM, in2 := #Minutes, out => #Flow_S)
      { S7_Templates := "SrcType := Real"; S7_GenerateENO := "TRUE" } Mul(in1 := #Flow_S, in2 := #Weight, out => #Flow_Speed)
   END_RUNG
   RUNG wire#w1
      { S7_Templates := "SrcType := Real" } EQ_Contact(in1 := #Filter.Median, in2 := 0.0)
      Move(in := 0.0, out1 => #Flow_S, out2 => #Flow_Speed)
   END_RUNG
   // the same network as SCL:
   IF NOT #Mode AND (#Filter.Median > 0.0) THEN
       #Flow_DTM := #Minutes / #Filter.Median;
       #Flow_S := #Flow_DTM * #Minutes;
       #Flow_Speed := #Flow_S * #Weight;
   END_IF;
   IF NOT #Mode AND (#Filter.Median = 0.0) THEN
       #Flow_S := 0.0;
       #Flow_Speed := 0.0;
   END_IF;
END_REGION

REGION Network 8: Рассчёт скорости потока по частому импульсному сигналу
   RUNG wire#powerrail
      P_Contact(operand := #pulse, bit := #pos[4])
      Move(in := 0.0, out1 => #Flow_DT)
      Not()
      I_Contact( #Mode )
      Contact( #Fast_Mode )
      wire#w1
      Contact( #Start )
      Add(in1 := #Flow_DT, in2 := #clock, out => #Flow_DT)
   END_RUNG
   RUNG wire#w1
      I_Contact( #Start )
      wire#w2
      Move(in := 0.0, out1 => #Flow_Speed)
   END_RUNG
   RUNG wire#w1
      Contact( #TimeControl."Exit" )
   END_RUNG wire#w2
   // the same network as SCL:
   #_w1 := #pulse AND NOT #pos[4];   // rising edge of #pulse
   #pos[4] := #pulse;
   IF #_w1 THEN #Flow_DT := 0.0; END_IF;
   #_w2 := NOT #_w1 AND NOT #Mode AND #Fast_Mode;
   IF #_w2 AND #Start THEN #Flow_DT := #Flow_DT + #clock; END_IF;
   IF #_w2 AND (NOT #Start OR #TimeControl."Exit") THEN #Flow_Speed := 0.0; END_IF;
END_REGION

REGION Network 9: Рассчёт скорости потока по аналоговому сигналу
   RUNG wire#powerrail
      Contact( #Mode )
      Move(in := #Weight_S, out1 => #Flow_S)
   END_RUNG
   // the same network as SCL:
   IF #Mode THEN #Flow_S := #Weight_S; END_IF;
END_REGION

REGION Network 10: Время сохранения суточного расхода
   RUNG wire#powerrail
      { S7_Templates := "SrcType := Int" } NE_Contact(in1 := #Day, in2 := "Time_SYS_DB".Time_Now.Day)
      S_Coil( #SaveDay )
   END_RUNG
   // the same network as SCL:
   IF #Day <> "Time_SYS_DB".Time_Now.Day THEN #SaveDay := TRUE; END_IF;
END_REGION

REGION Network 11: Сохранить данные за сеанс
   RUNG wire#powerrail
      Contact( #Save )
      { S7_GenerateENO := "TRUE" } Move(in := #Seans, out1 => #Seans_Last)
      { S7_GenerateENO := "TRUE" } Move(in := 0.0, out1 => #Seans)
      R_Coil( #Save )
   END_RUNG
   // the same network as SCL:
   // ENO of a box is taken as its EN; it also drops when the box reports an error
   IF #Save THEN
       #Seans_Last := #Seans;
       #Seans := 0.0;
       #Save := FALSE;
   END_IF;
END_REGION

REGION Network 12: Сохранить данные за сутки
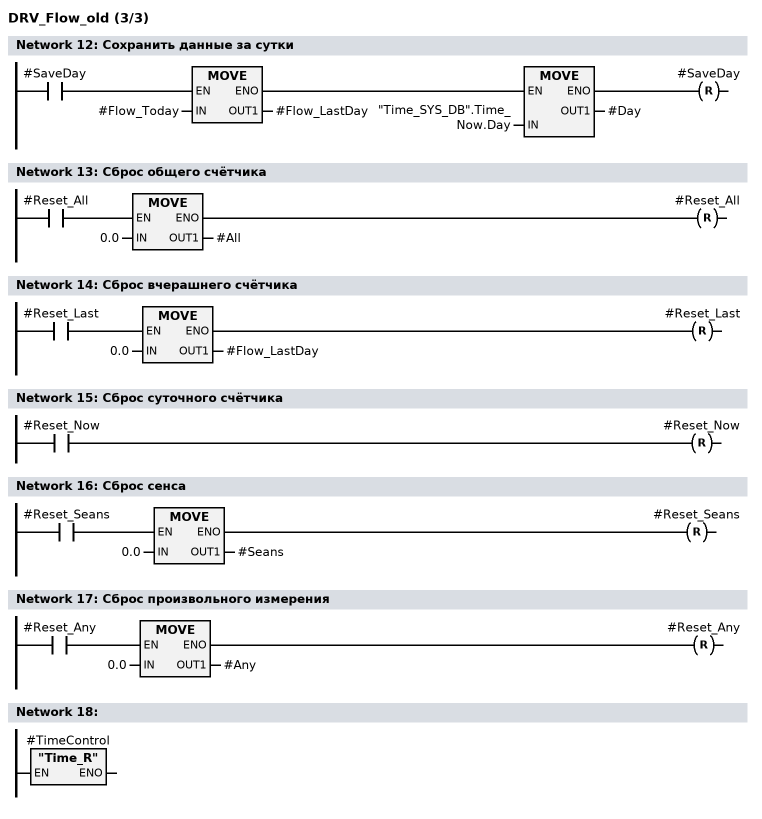
   RUNG wire#powerrail
      Contact( #SaveDay )
      { S7_GenerateENO := "TRUE" } Move(in := #Flow_Today, out1 => #Flow_LastDay)
      { S7_GenerateENO := "TRUE" } Move(in := "Time_SYS_DB".Time_Now.Day, out1 => #Day)
      R_Coil( #SaveDay )
   END_RUNG
   // the same network as SCL:
   // ENO of a box is taken as its EN; it also drops when the box reports an error
   IF #SaveDay THEN
       #Flow_LastDay := #Flow_Today;
       #Day := "Time_SYS_DB".Time_Now.Day;
       #SaveDay := FALSE;
   END_IF;
END_REGION

REGION Network 13: Сброс общего счётчика
   RUNG wire#powerrail
      Contact( #Reset_All )
      { S7_GenerateENO := "TRUE" } Move(in := 0.0, out1 => #All)
      R_Coil( #Reset_All )
   END_RUNG
   // the same network as SCL:
   // ENO of a box is taken as its EN; it also drops when the box reports an error
   IF #Reset_All THEN
       #All := 0.0;
       #Reset_All := FALSE;
   END_IF;
END_REGION

REGION Network 14: Сброс вчерашнего счётчика
   RUNG wire#powerrail
      Contact( #Reset_Last )
      { S7_GenerateENO := "TRUE" } Move(in := 0.0, out1 => #Flow_LastDay)
      R_Coil( #Reset_Last )
   END_RUNG
   // the same network as SCL:
   // ENO of a box is taken as its EN; it also drops when the box reports an error
   IF #Reset_Last THEN
       #Flow_LastDay := 0.0;
       #Reset_Last := FALSE;
   END_IF;
END_REGION

REGION Network 15: Сброс суточного счётчика
   RUNG wire#powerrail
      Contact( #Reset_Now )
      R_Coil( #Reset_Now )
   END_RUNG
   // the same network as SCL:
   IF #Reset_Now THEN #Reset_Now := FALSE; END_IF;
END_REGION

REGION Network 16: Сброс сенса
   RUNG wire#powerrail
      Contact( #Reset_Seans )
      { S7_GenerateENO := "TRUE" } Move(in := 0.0, out1 => #Seans)
      R_Coil( #Reset_Seans )
   END_RUNG
   // the same network as SCL:
   // ENO of a box is taken as its EN; it also drops when the box reports an error
   IF #Reset_Seans THEN
       #Seans := 0.0;
       #Reset_Seans := FALSE;
   END_IF;
END_REGION

REGION Network 17: Сброс произвольного измерения
   RUNG wire#powerrail
      Contact( #Reset_Any )
      { S7_GenerateENO := "TRUE" } Move(in := 0.0, out1 => #Any)
      R_Coil( #Reset_Any )
   END_RUNG
   // the same network as SCL:
   // ENO of a box is taken as its EN; it also drops when the box reports an error
   IF #Reset_Any THEN
       #Any := 0.0;
       #Reset_Any := FALSE;
   END_IF;
END_REGION

REGION Network 18
   RUNG wire#powerrail
      #TimeControl()
   END_RUNG
   // the same network as SCL:
   #TimeControl();   // "Time_R"
END_REGION
END_FUNCTION_BLOCK

FUNCTION_BLOCK "Block_Pump"   // FB13, LAD
{ S7_Optimized_Access := 'TRUE' }
VERSION : 0.1
// stored: AutoNumber true, IsIECCheckEnabled false, IsRetainMemResEnabled false, MemoryReserve 100, SetENOAutomatically false, UDAEnableTagReadback false
   VAR_INPUT
      All_Lines : Int;
      Status_Pump : Int;
   END_VAR
   VAR_OUTPUT
      Alarm : Bool;
      CMD_Alarm : Bool;
      SP_Result : Real;
   END_VAR
   VAR_IN_OUT
      Start_A : Bool;
   END_VAR
   VAR RETAIN
      PUMP_NUMBER : Int;
      Reserv { S7_SetPoint := 'True'} : Bool;
   END_VAR
   VAR
      Start_Main : Bool;
      Start_Reserv : Bool;
      REQ : Bool;
      REQ_Reserv : Bool;   // Запрос резерва с панели
      pos : Array[0..15] of Bool;
      Events : Word;
   END_VAR
   VAR RETAIN
      Line_Main { S7_SetPoint := 'True'} : Int;
      Line_Reserv { S7_SetPoint := 'True'} : Int;
   END_VAR
   VAR
      T_events : Struct
         SP { ExternalAccessible := 'False'; ExternalVisible := 'False'; ExternalWritable := 'False'} : Int := 3;   // Уставка
         Now { ExternalAccessible := 'False'; ExternalVisible := 'False'; ExternalWritable := 'False'} : Int;   // Текущий счёт
         "Exit" { ExternalAccessible := 'False'; ExternalVisible := 'False'; ExternalWritable := 'False'} : Bool;   // Счёт завершён
         Start { ExternalAccessible := 'False'; ExternalVisible := 'False'; ExternalWritable := 'False'} : Bool;   // Запуск
         Pause { ExternalAccessible := 'False'; ExternalVisible := 'False'; ExternalWritable := 'False'} : Bool;   // Пауза
         Reset { ExternalAccessible := 'False'; ExternalVisible := 'False'; ExternalWritable := 'False'} : Bool;   // Сброс таймера
      END_STRUCT;
   END_VAR
   VAR_TEMP
      ev : Bool;
   END_VAR
   VAR_TEMP   // added for the SCL form of the ladder/FBD networks
      _w1 : Bool;
      _w2 : Bool;
      _w3 : Bool;
      _w4 : Bool;
      _w5 : Bool;
      _w6 : Bool;
      _w7 : Bool;
      _w8 : Bool;
      _w9 : Bool;
      _w10 : Bool;
   END_VAR
BEGIN

REGION Network 1
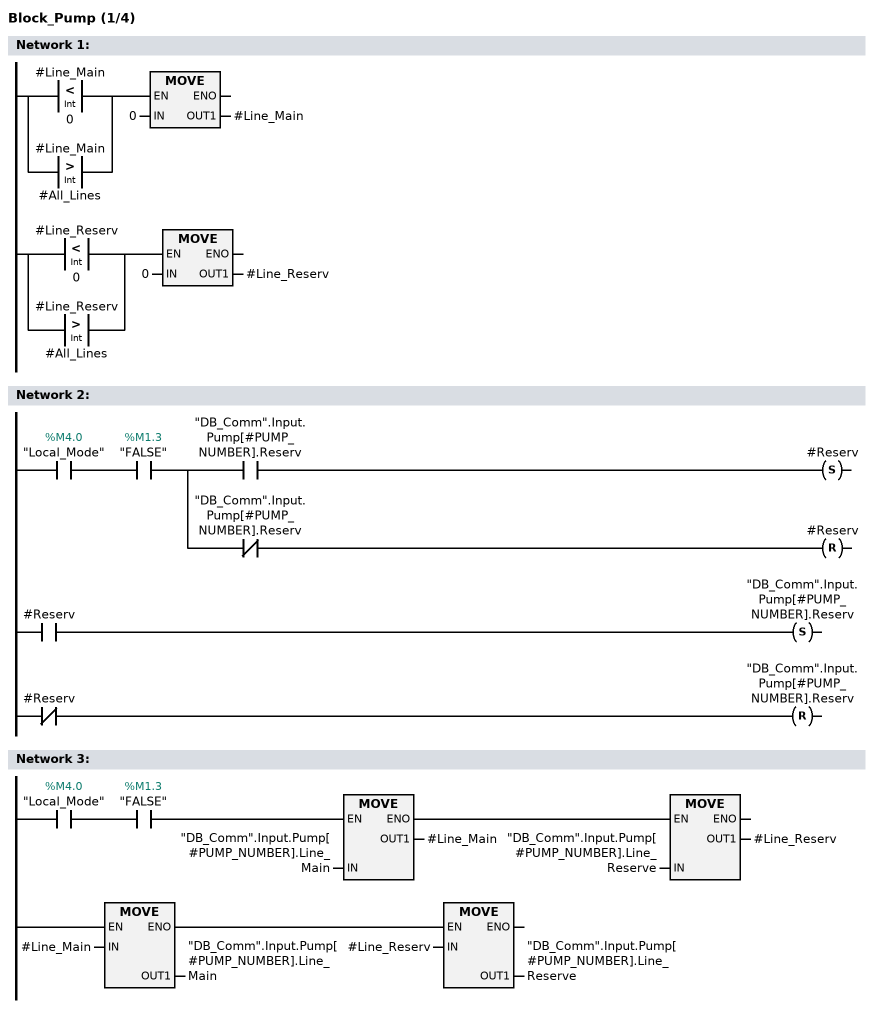
   RUNG wire#powerrail
      { S7_Templates := "SrcType := Int" } LT_Contact(in1 := #Line_Main, in2 := 0)
      wire#w1
      Move(in := 0, out1 => #Line_Main)
   END_RUNG
   RUNG wire#powerrail
      { S7_Templates := "SrcType := Int" } GT_Contact(in1 := #Line_Main, in2 := #All_Lines)
   END_RUNG wire#w1
   RUNG wire#powerrail
      { S7_Templates := "SrcType := Int" } LT_Contact(in1 := #Line_Reserv, in2 := 0)
      wire#w2
      Move(in := 0, out1 => #Line_Reserv)
   END_RUNG
   RUNG wire#powerrail
      { S7_Templates := "SrcType := Int" } GT_Contact(in1 := #Line_Reserv, in2 := #All_Lines)
   END_RUNG wire#w2
   // the same network as SCL:
   IF (#Line_Main < 0) OR (#Line_Main > #All_Lines) THEN #Line_Main := 0; END_IF;
   IF (#Line_Reserv < 0) OR (#Line_Reserv > #All_Lines) THEN #Line_Reserv := 0; END_IF;
END_REGION

REGION Network 2
   RUNG wire#powerrail
      Contact( "Local_Mode" )
      Contact( "FALSE" )
      wire#w1
      Contact( "DB_Comm".Input.Pump[#PUMP_NUMBER].Reserv )
      S_Coil( #Reserv )
   END_RUNG
   RUNG wire#w1
      I_Contact( "DB_Comm".Input.Pump[#PUMP_NUMBER].Reserv )
      R_Coil( #Reserv )
   END_RUNG
   RUNG wire#powerrail
      Contact( #Reserv )
      S_Coil( "DB_Comm".Input.Pump[#PUMP_NUMBER].Reserv )
   END_RUNG
   RUNG wire#powerrail
      I_Contact( #Reserv )
      R_Coil( "DB_Comm".Input.Pump[#PUMP_NUMBER].Reserv )
   END_RUNG
   // the same network as SCL:
   #_w1 := "Local_Mode" AND "FALSE";
   IF #_w1 AND "DB_Comm".Input.Pump[#PUMP_NUMBER].Reserv THEN #Reserv := TRUE; END_IF;
   IF #_w1 AND NOT "DB_Comm".Input.Pump[#PUMP_NUMBER].Reserv THEN #Reserv := FALSE; END_IF;
   IF #Reserv THEN "DB_Comm".Input.Pump[#PUMP_NUMBER].Reserv := TRUE; END_IF;
   IF NOT #Reserv THEN "DB_Comm".Input.Pump[#PUMP_NUMBER].Reserv := FALSE; END_IF;
END_REGION

REGION Network 3
   RUNG wire#powerrail
      Contact( "Local_Mode" )
      Contact( "FALSE" )
      Move(in := "DB_Comm".Input.Pump[#PUMP_NUMBER].Line_Main, out1 => #Line_Main)
      Move(in := "DB_Comm".Input.Pump[#PUMP_NUMBER].Line_Reserve, out1 => #Line_Reserv)
   END_RUNG
   RUNG wire#powerrail
      Move(in := #Line_Main, out1 => "DB_Comm".Input.Pump[#PUMP_NUMBER].Line_Main)
      Move(in := #Line_Reserv, out1 => "DB_Comm".Input.Pump[#PUMP_NUMBER].Line_Reserve)
   END_RUNG
   // the same network as SCL:
   IF "Local_Mode" AND "FALSE" THEN
       #Line_Main := "DB_Comm".Input.Pump[#PUMP_NUMBER].Line_Main;
       #Line_Reserv := "DB_Comm".Input.Pump[#PUMP_NUMBER].Line_Reserve;
   END_IF;
   "DB_Comm".Input.Pump[#PUMP_NUMBER].Line_Main := #Line_Main;
   "DB_Comm".Input.Pump[#PUMP_NUMBER].Line_Reserve := #Line_Reserv;
END_REGION

REGION Network 4: Основной насос
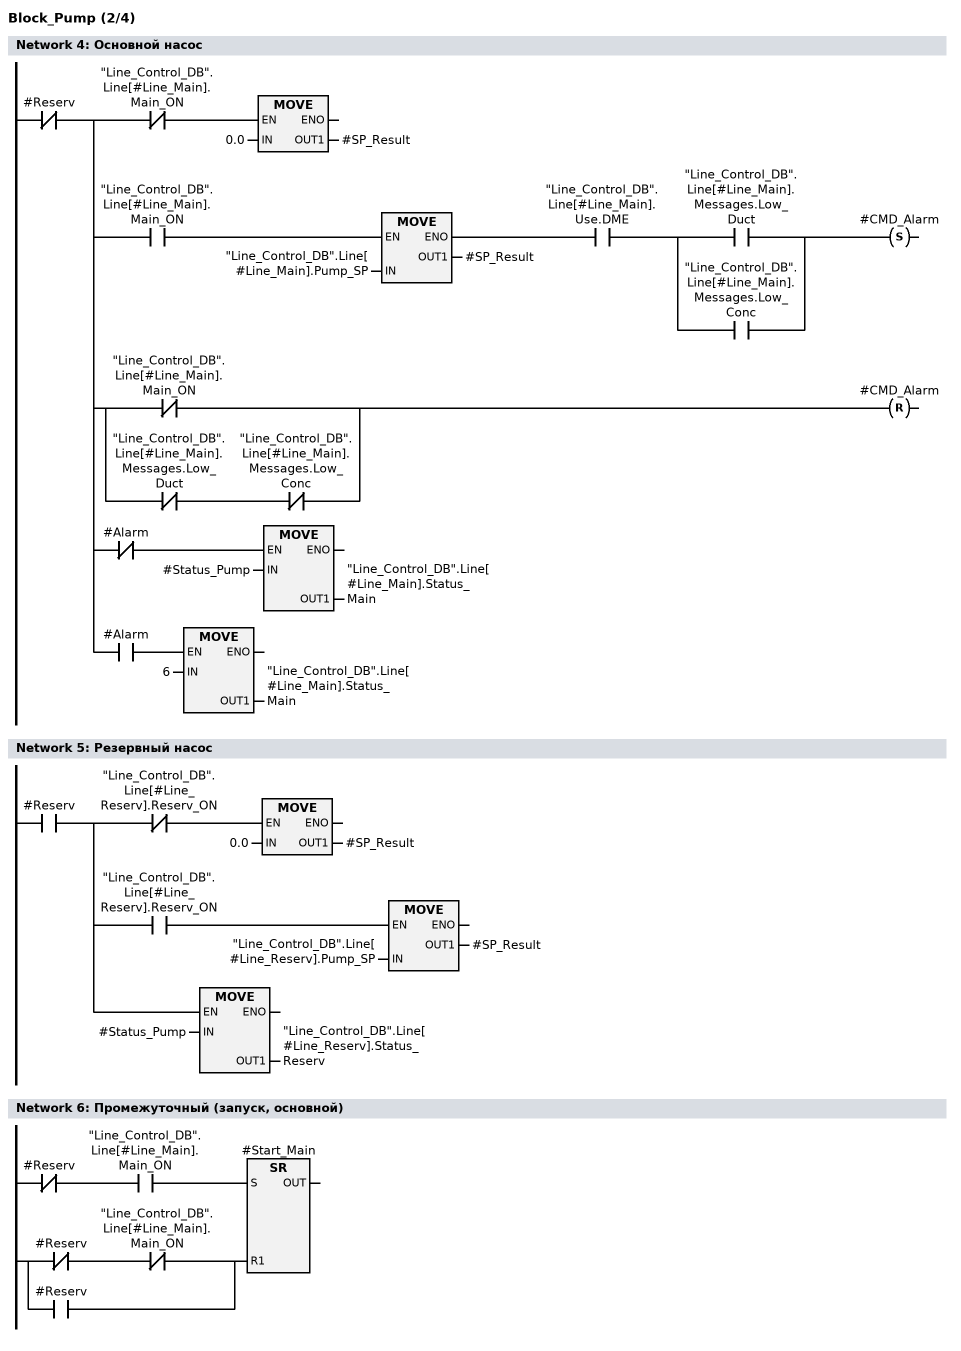
   RUNG wire#powerrail
      I_Contact( #Reserv )
      wire#w1
      I_Contact( "Line_Control_DB".Line[#Line_Main].Main_ON )
      Move(in := 0.0, out1 => #SP_Result)
   END_RUNG
   RUNG wire#w1
      Contact( "Line_Control_DB".Line[#Line_Main].Main_ON )
      Move(in := "Line_Control_DB".Line[#Line_Main].Pump_SP, out1 => #SP_Result)
      Contact( "Line_Control_DB".Line[#Line_Main].Use.DME )
      wire#w2
      Contact( "Line_Control_DB".Line[#Line_Main].Messages.Low_Duct )
      wire#w3
      S_Coil( #CMD_Alarm )
   END_RUNG
   RUNG wire#w2
      Contact( "Line_Control_DB".Line[#Line_Main].Messages.Low_Conc )
   END_RUNG wire#w3
   RUNG wire#w1
      I_Contact( "Line_Control_DB".Line[#Line_Main].Main_ON )
      wire#w4
      R_Coil( #CMD_Alarm )
   END_RUNG
   RUNG wire#w1
      I_Contact( "Line_Control_DB".Line[#Line_Main].Messages.Low_Duct )
      I_Contact( "Line_Control_DB".Line[#Line_Main].Messages.Low_Conc )
   END_RUNG wire#w4
   RUNG wire#w1
      I_Contact( #Alarm )
      Move(in := #Status_Pump, out1 => "Line_Control_DB".Line[#Line_Main].Status_Main)
   END_RUNG
   RUNG wire#w1
      Contact( #Alarm )
      Move(in := 6, out1 => "Line_Control_DB".Line[#Line_Main].Status_Main)
   END_RUNG
   // the same network as SCL:
   IF NOT #Reserv AND NOT "Line_Control_DB".Line[#Line_Main].Main_ON THEN #SP_Result := 0.0; END_IF;
   #_w1 := NOT #Reserv AND "Line_Control_DB".Line[#Line_Main].Main_ON;
   IF #_w1 THEN #SP_Result := "Line_Control_DB".Line[#Line_Main].Pump_SP; END_IF;
   IF #_w1 AND "Line_Control_DB".Line[#Line_Main].Use.DME AND ("Line_Control_DB".Line[#Line_Main].Messages.Low_Duct OR "Line_Control_DB".Line[#Line_Main].Messages.Low_Conc) THEN
       #CMD_Alarm := TRUE;
   END_IF;
   IF NOT #Reserv AND (NOT "Line_Control_DB".Line[#Line_Main].Main_ON OR (NOT "Line_Control_DB".Line[#Line_Main].Messages.Low_Duct AND NOT "Line_Control_DB".Line[#Line_Main].Messages.Low_Conc)) THEN
       #CMD_Alarm := FALSE;
   END_IF;
   IF NOT #Reserv AND NOT #Alarm THEN "Line_Control_DB".Line[#Line_Main].Status_Main := #Status_Pump; END_IF;
   IF NOT #Reserv AND #Alarm THEN "Line_Control_DB".Line[#Line_Main].Status_Main := 6; END_IF;
END_REGION

REGION Network 5: Резервный насос
   RUNG wire#powerrail
      Contact( #Reserv )
      wire#w1
      I_Contact( "Line_Control_DB".Line[#Line_Reserv].Reserv_ON )
      Move(in := 0.0, out1 => #SP_Result)
   END_RUNG
   RUNG wire#w1
      Contact( "Line_Control_DB".Line[#Line_Reserv].Reserv_ON )
      Move(in := "Line_Control_DB".Line[#Line_Reserv].Pump_SP, out1 => #SP_Result)
   END_RUNG
   RUNG wire#w1
      Move(in := #Status_Pump, out1 => "Line_Control_DB".Line[#Line_Reserv].Status_Reserv)
   END_RUNG
   // the same network as SCL:
   IF #Reserv AND NOT "Line_Control_DB".Line[#Line_Reserv].Reserv_ON THEN #SP_Result := 0.0; END_IF;
   IF #Reserv AND "Line_Control_DB".Line[#Line_Reserv].Reserv_ON THEN
       #SP_Result := "Line_Control_DB".Line[#Line_Reserv].Pump_SP;
   END_IF;
   IF #Reserv THEN "Line_Control_DB".Line[#Line_Reserv].Status_Reserv := #Status_Pump; END_IF;
END_REGION

REGION Network 6: Промежуточный (запуск, основной)
   RUNG wire#powerrail
      I_Contact( #Reserv )
      Contact( "Line_Control_DB".Line[#Line_Main].Main_ON )
      S_SR(operand := #Start_Main, r1 := wire#w1)
   END_RUNG
   RUNG wire#powerrail
      I_Contact( #Reserv )
      I_Contact( "Line_Control_DB".Line[#Line_Main].Main_ON )
   END_RUNG wire#w1
   RUNG wire#powerrail
      Contact( #Reserv )
   END_RUNG wire#w1
   // the same network as SCL:
   IF NOT #Reserv AND "Line_Control_DB".Line[#Line_Main].Main_ON THEN
       #Start_Main := TRUE;   // SR flip-flop
   END_IF;
   IF (NOT #Reserv AND NOT "Line_Control_DB".Line[#Line_Main].Main_ON) OR #Reserv THEN
       #Start_Main := FALSE;
   END_IF;
END_REGION

REGION Network 7: Промежуточный (запуск, резервный)
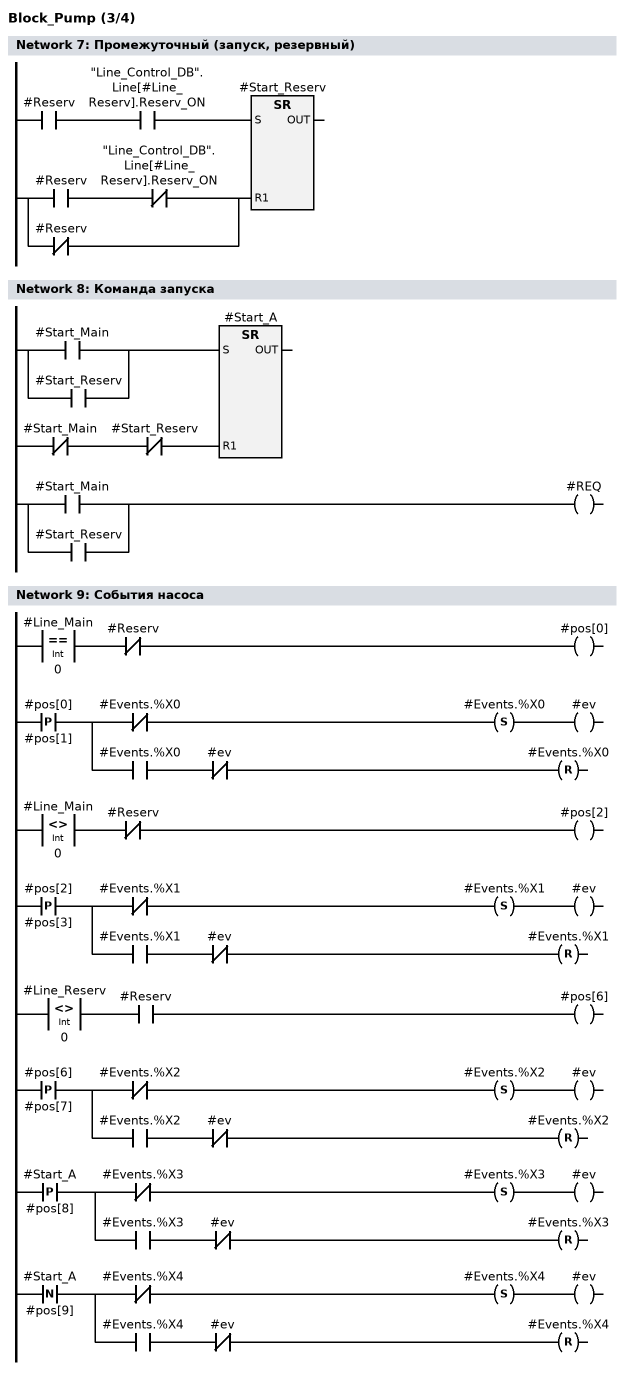
   RUNG wire#powerrail
      Contact( #Reserv )
      Contact( "Line_Control_DB".Line[#Line_Reserv].Reserv_ON )
      S_SR(operand := #Start_Reserv, r1 := wire#w1)
   END_RUNG
   RUNG wire#powerrail
      Contact( #Reserv )
      I_Contact( "Line_Control_DB".Line[#Line_Reserv].Reserv_ON )
   END_RUNG wire#w1
   RUNG wire#powerrail
      I_Contact( #Reserv )
   END_RUNG wire#w1
   // the same network as SCL:
   IF #Reserv AND "Line_Control_DB".Line[#Line_Reserv].Reserv_ON THEN
       #Start_Reserv := TRUE;   // SR flip-flop
   END_IF;
   IF (#Reserv AND NOT "Line_Control_DB".Line[#Line_Reserv].Reserv_ON) OR NOT #Reserv THEN
       #Start_Reserv := FALSE;
   END_IF;
END_REGION

REGION Network 8: Команда запуска
   RUNG wire#powerrail
      Contact( #Start_Main )
      wire#w1
      S_SR(operand := #Start_A, r1 := wire#w2)
   END_RUNG
   RUNG wire#powerrail
      Contact( #Start_Reserv )
   END_RUNG wire#w1
   RUNG wire#powerrail
      I_Contact( #Start_Main )
      I_Contact( #Start_Reserv )
   END_RUNG wire#w2
   RUNG wire#powerrail
      Contact( #Start_Main )
      wire#w3
      Coil( #REQ )
   END_RUNG
   RUNG wire#powerrail
      Contact( #Start_Reserv )
   END_RUNG wire#w3
   // the same network as SCL:
   IF #Start_Main OR #Start_Reserv THEN
       #Start_A := TRUE;   // SR flip-flop
   END_IF;
   IF NOT #Start_Main AND NOT #Start_Reserv THEN #Start_A := FALSE; END_IF;
   #REQ := #Start_Main OR #Start_Reserv;
END_REGION

REGION Network 9: События насоса
   RUNG wire#powerrail
      { S7_Templates := "SrcType := Int" } EQ_Contact(in1 := #Line_Main, in2 := 0)
      I_Contact( #Reserv )
      Coil( #pos[0] )
   END_RUNG
   RUNG wire#powerrail
      P_Contact(operand := #pos[0], bit := #pos[1])
      wire#w1
      I_Contact( #Events.%X0 )
      S_Coil( #Events.%X0 )
      Coil( #ev )
   END_RUNG
   RUNG wire#w1
      Contact( #Events.%X0 )
      I_Contact( #ev )
      R_Coil( #Events.%X0 )
   END_RUNG
   RUNG wire#powerrail
      { S7_Templates := "SrcType := Int" } NE_Contact(in1 := #Line_Main, in2 := 0)
      I_Contact( #Reserv )
      Coil( #pos[2] )
   END_RUNG
   RUNG wire#powerrail
      P_Contact(operand := #pos[2], bit := #pos[3])
      wire#w2
      I_Contact( #Events.%X1 )
      S_Coil( #Events.%X1 )
      Coil( #ev )
   END_RUNG
   RUNG wire#w2
      Contact( #Events.%X1 )
      I_Contact( #ev )
      R_Coil( #Events.%X1 )
   END_RUNG
   RUNG wire#powerrail
      { S7_Templates := "SrcType := Int" } NE_Contact(in1 := #Line_Reserv, in2 := 0)
      Contact( #Reserv )
      Coil( #pos[6] )
   END_RUNG
   RUNG wire#powerrail
      P_Contact(operand := #pos[6], bit := #pos[7])
      wire#w3
      I_Contact( #Events.%X2 )
      S_Coil( #Events.%X2 )
      Coil( #ev )
   END_RUNG
   RUNG wire#w3
      Contact( #Events.%X2 )
      I_Contact( #ev )
      R_Coil( #Events.%X2 )
   END_RUNG
   RUNG wire#powerrail
      P_Contact(operand := #Start_A, bit := #pos[8])
      wire#w4
      I_Contact( #Events.%X3 )
      S_Coil( #Events.%X3 )
      Coil( #ev )
   END_RUNG
   RUNG wire#w4
      Contact( #Events.%X3 )
      I_Contact( #ev )
      R_Coil( #Events.%X3 )
   END_RUNG
   RUNG wire#powerrail
      N_Contact(operand := #Start_A, bit := #pos[9])
      wire#w5
      I_Contact( #Events.%X4 )
      S_Coil( #Events.%X4 )
      Coil( #ev )
   END_RUNG
   RUNG wire#w5
      Contact( #Events.%X4 )
      I_Contact( #ev )
      R_Coil( #Events.%X4 )
   END_RUNG
   // the same network as SCL:
   #pos[0] := (#Line_Main = 0) AND NOT #Reserv;
   #_w1 := #pos[0] AND NOT #pos[1];   // rising edge of #pos[0]
   #pos[1] := #pos[0];
   #_w2 := #_w1 AND NOT #Events.%X0;
   IF #_w2 THEN #Events.%X0 := TRUE; END_IF;
   #ev := #_w2;
   IF #_w1 AND #Events.%X0 AND NOT #ev THEN #Events.%X0 := FALSE; END_IF;
   #pos[2] := (#Line_Main <> 0) AND NOT #Reserv;
   #_w3 := #pos[2] AND NOT #pos[3];   // rising edge of #pos[2]
   #pos[3] := #pos[2];
   #_w4 := #_w3 AND NOT #Events.%X1;
   IF #_w4 THEN #Events.%X1 := TRUE; END_IF;
   #ev := #_w4;
   IF #_w3 AND #Events.%X1 AND NOT #ev THEN #Events.%X1 := FALSE; END_IF;
   #pos[6] := (#Line_Reserv <> 0) AND #Reserv;
   #_w5 := #pos[6] AND NOT #pos[7];   // rising edge of #pos[6]
   #pos[7] := #pos[6];
   #_w6 := #_w5 AND NOT #Events.%X2;
   IF #_w6 THEN #Events.%X2 := TRUE; END_IF;
   #ev := #_w6;
   IF #_w5 AND #Events.%X2 AND NOT #ev THEN #Events.%X2 := FALSE; END_IF;
   #_w7 := #Start_A AND NOT #pos[8];   // rising edge of #Start_A
   #pos[8] := #Start_A;
   #_w8 := #_w7 AND NOT #Events.%X3;
   IF #_w8 THEN #Events.%X3 := TRUE; END_IF;
   #ev := #_w8;
   IF #_w7 AND #Events.%X3 AND NOT #ev THEN #Events.%X3 := FALSE; END_IF;
   #_w9 := NOT #Start_A AND #pos[9];   // falling edge of #Start_A
   #pos[9] := #Start_A;
   #_w10 := #_w9 AND NOT #Events.%X4;
   IF #_w10 THEN #Events.%X4 := TRUE; END_IF;
   #ev := #_w10;
   IF #_w9 AND #Events.%X4 AND NOT #ev THEN #Events.%X4 := FALSE; END_IF;
END_REGION

REGION Network 10
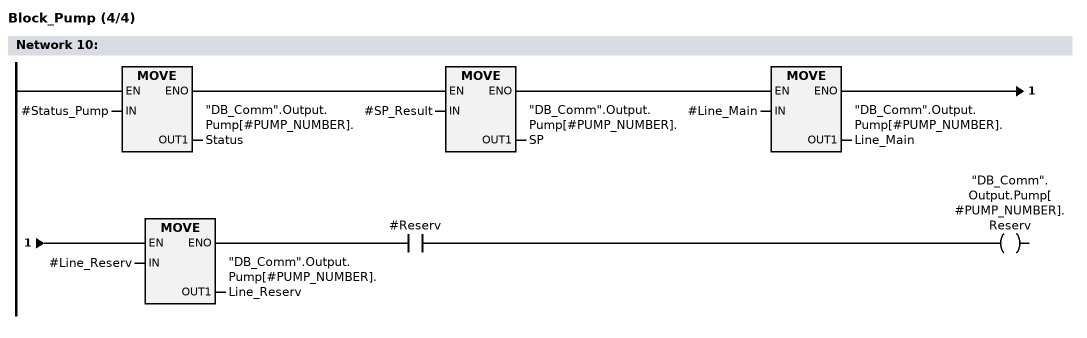
   RUNG wire#powerrail
      Move(in := #Status_Pump, out1 => "DB_Comm".Output.Pump[#PUMP_NUMBER].Status)
      Move(in := #SP_Result, out1 => "DB_Comm".Output.Pump[#PUMP_NUMBER].SP)
      Move(in := #Line_Main, out1 => "DB_Comm".Output.Pump[#PUMP_NUMBER].Line_Main)
      Move(in := #Line_Reserv, out1 => "DB_Comm".Output.Pump[#PUMP_NUMBER].Line_Reserv)
      Contact( #Reserv )
      Coil( "DB_Comm".Output.Pump[#PUMP_NUMBER].Reserv )
   END_RUNG
   // the same network as SCL:
   "DB_Comm".Output.Pump[#PUMP_NUMBER].Status := #Status_Pump;
   "DB_Comm".Output.Pump[#PUMP_NUMBER].SP := #SP_Result;
   "DB_Comm".Output.Pump[#PUMP_NUMBER].Line_Main := #Line_Main;
   "DB_Comm".Output.Pump[#PUMP_NUMBER].Line_Reserv := #Line_Reserv;
   "DB_Comm".Output.Pump[#PUMP_NUMBER].Reserv := #Reserv;
END_REGION
END_FUNCTION_BLOCK

FUNCTION "Report_Line_FC" : Void
{ S7_Optimized_Access := 'TRUE' }
VERSION : 0.1
   VAR_INPUT 
      Reset : Bool;
      Line : Int;
   END_VAR

   VAR_IN_OUT 
      Report : Struct
         Last_Day : Int;
         Last_Date : Int;
         Last_Month : Int;
         RM_1 : Real;   // Расходомер 1
         RM_2 : Real;   // Расходомер 2
         D_Mid : Real;   // Средняя доза за сутки
         Flow : Real;   // Общая труба (куда происходит дозация)
         Days : Array[1..7] of "Line_Report";
         cnt : Int;
         cnt_x : Int;
      END_STRUCT;
      cnt : Int;
      cnt_x : Int;
   END_VAR

   VAR_TEMP 
      x : Int;
   END_VAR


BEGIN
	#Report.RM_1 := "Line_Control_DB".Line[#Line].FlowMeter_1.Flow_Today;
	#Report.RM_2 := "Line_Control_DB".Line[#Line].FlowMeter_2.Flow_Today;
	IF "pulse_1s" THEN
	    #Report.Flow := #Report.Flow + "Line_Control_DB".Line[#Line].Flow_s;
	END_IF;
	IF "Line_Control_DB".Line[#Line].D_Num <> 0 THEN
	    #Report.D_Mid := "Line_Control_DB".Line[#Line].D_Sum / "Line_Control_DB".Line[#Line].D_Num;
	ELSE
	    #Report.D_Mid := 0.0;
	END_IF;
	//сдвиг по дням недели
	//
	
	IF #Report.Last_Date <> "Time_SYS_DB".Time_Now.Day THEN
	    
	    IF #cnt <= 0 THEN
	        #cnt := 7;
	    END_IF;
	    
	    IF #cnt > 1 THEN
	        #cnt_x := #cnt - 1;
	        #Report.Days[#cnt] :=#Report.Days[#cnt_x];
	        #cnt := #cnt_x;
	    END_IF;
	    
	    IF #cnt = 1 THEN
	            //#Comm_Days := #Report.Days[1];
	            
	            
	            #Report.Days[1].RM_1 := #Report.RM_1;
	            #Report.Days[1].RM_2 := #Report.RM_2;
	            #Report.Days[1].D_Mid :=#Report.D_Mid;
	            #Report.Days[1].Flow :=#Report.Flow;
	            #Report.Days[1].Day :=#Report.Last_Date;
	            #Report.Days[1].Month :=#Report.Last_Month;
	            #Report.Days[1].WeekDay :=#Report.Last_Day;
	            
	            #Report.RM_1 := 0.0;
	            #Report.RM_2 := 0.0;
	            #Report.D_Mid := 0.0;
	            #Report.Flow := 0.0;
	            
	            #Report.Last_Month :="Time_SYS_DB".Time_Now.Month;
	            #Report.Last_Day :="Time_SYS_DB".Time_Now.Weekday;
	            #Report.Last_Date :="Time_SYS_DB".Time_Now.Day;
	            
	            "Line_Control_DB".Line[#Line].D_Sum := 0.0;
	            "Line_Control_DB".Line[#Line].D_Num := 0.0;
	            "Line_Control_DB".Line[#Line].FlowMeter_1.Flow_Today := 0.0;
	            "Line_Control_DB".Line[#Line].FlowMeter_2.Flow_Today := 0.0;
	    END_IF;
	END_IF;
	
	    
	    IF #Report.Last_Date ="Time_SYS_DB".Time_Now.Day THEN
	        #cnt := 7;
	    END_IF;
	    
	    IF #Reset THEN
	        FOR #x := 1 TO 7 DO
	            #Report.Days[#x].RM_1 := 0.0;
	            #Report.Days[#x].RM_2 := 0.0;
	            #Report.Days[#x].D_Mid := 0.0;
	            #Report.Days[#x].Flow := 0.0;
	            #Report.Days[#x].Day := 0;
	            #Report.Days[#x].Month := 0;
	            #Report.Days[#x].WeekDay := 0;
	            ;
	        END_FOR;
	    END_IF;
	    
	
END_FUNCTION

FUNCTION_BLOCK "Smena"   // FB17, LAD
{ S7_Optimized_Access := 'FALSE' }
VERSION : 0.1
// stored: AutoNumber true, IsIECCheckEnabled false, SetENOAutomatically false, UDAEnableTagReadback false
   VAR DB_SPECIFIC
      ON_1 : Struct
         Use : Bool;
         H : Int;
         "M" : Int;
      END_STRUCT;
      ON_2 : Struct
         Use : Bool;
         H : Int;
         "M" : Int;
      END_STRUCT;
      pos : Array[0..31] of Bool;
      Line_1 : Array[0..2] of Struct
         Water : Real;
         Reagent : Real;
      END_STRUCT;
      Line_2 : Array[0..2] of Struct
         Water : Real;
         Reagent : Real;
      END_STRUCT;
      "Time" : Array[0..2] of Struct
         Start_H : Int;
         Start_M : Int;
         "Date" : Int;
         Mounth : Int;
      END_STRUCT;
      Time_DTL : DTL;
   END_VAR
   VAR_TEMP
      x0 : Real;
      x1 : Real;
      x2 : Real;
      x3 : Real;
   END_VAR
   VAR_TEMP   // added for the SCL form of the ladder/FBD networks
      _w1 : Bool;
      _w2 : Bool;
   END_VAR
BEGIN

REGION Network 1: Первая запись
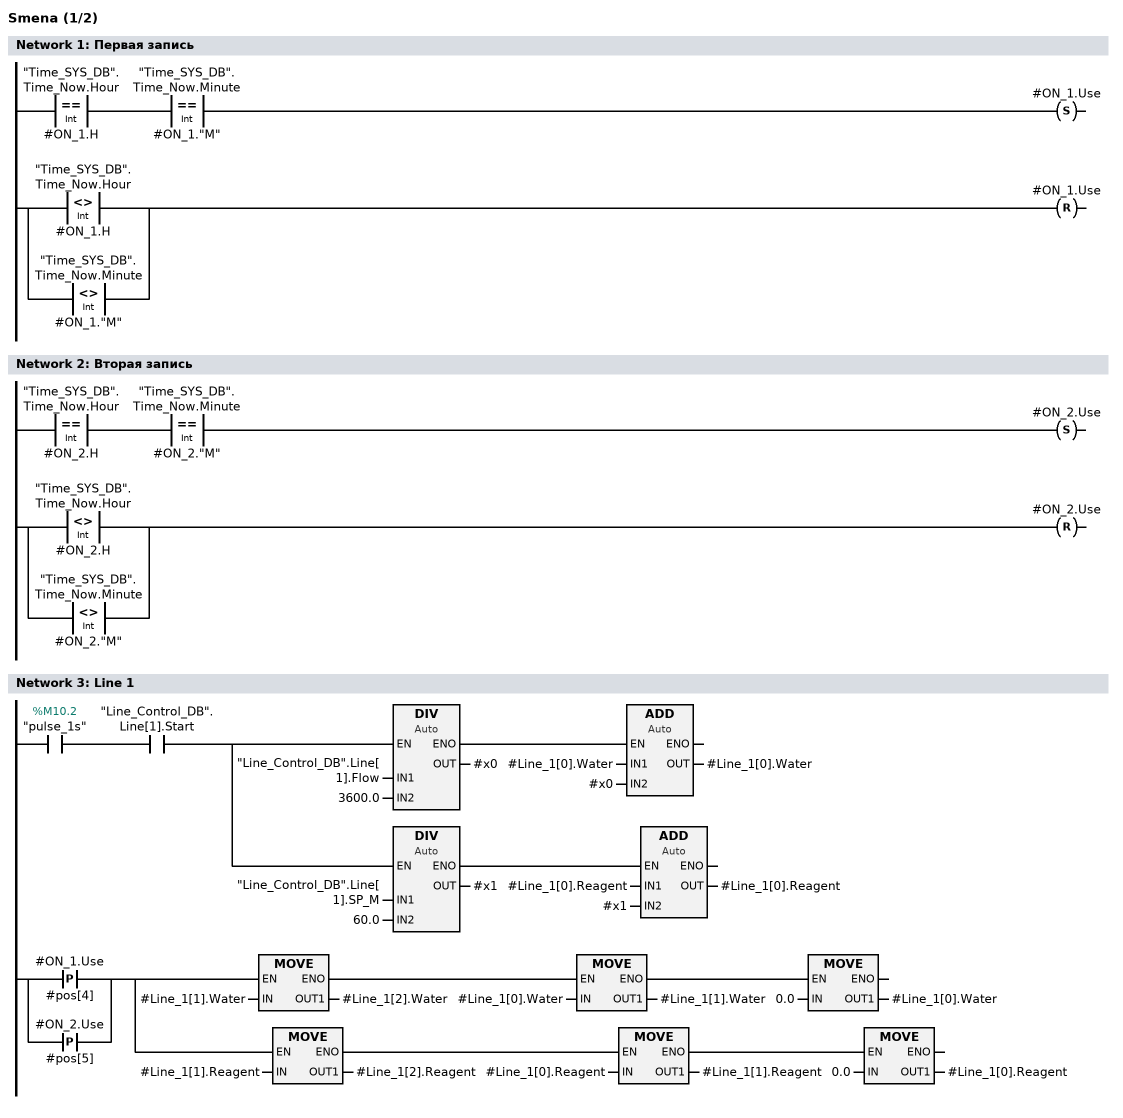
   RUNG wire#powerrail
      { S7_Templates := "SrcType := Int" } EQ_Contact(in1 := "Time_SYS_DB".Time_Now.Hour, in2 := #ON_1.H)
      { S7_Templates := "SrcType := Int" } EQ_Contact(in1 := "Time_SYS_DB".Time_Now.Minute, in2 := #ON_1."M")
      S_Coil( #ON_1.Use )
   END_RUNG
   RUNG wire#powerrail
      { S7_Templates := "SrcType := Int" } NE_Contact(in1 := "Time_SYS_DB".Time_Now.Hour, in2 := #ON_1.H)
      wire#w1
      R_Coil( #ON_1.Use )
   END_RUNG
   RUNG wire#powerrail
      { S7_Templates := "SrcType := Int" } NE_Contact(in1 := "Time_SYS_DB".Time_Now.Minute, in2 := #ON_1."M")
   END_RUNG wire#w1
   // the same network as SCL:
   IF ("Time_SYS_DB".Time_Now.Hour = #ON_1.H) AND ("Time_SYS_DB".Time_Now.Minute = #ON_1."M") THEN
       #ON_1.Use := TRUE;
   END_IF;
   IF ("Time_SYS_DB".Time_Now.Hour <> #ON_1.H) OR ("Time_SYS_DB".Time_Now.Minute <> #ON_1."M") THEN
       #ON_1.Use := FALSE;
   END_IF;
END_REGION

REGION Network 2: Вторая запись
   RUNG wire#powerrail
      { S7_Templates := "SrcType := Int" } EQ_Contact(in1 := "Time_SYS_DB".Time_Now.Hour, in2 := #ON_2.H)
      { S7_Templates := "SrcType := Int" } EQ_Contact(in1 := "Time_SYS_DB".Time_Now.Minute, in2 := #ON_2."M")
      S_Coil( #ON_2.Use )
   END_RUNG
   RUNG wire#powerrail
      { S7_Templates := "SrcType := Int" } NE_Contact(in1 := "Time_SYS_DB".Time_Now.Hour, in2 := #ON_2.H)
      wire#w1
      R_Coil( #ON_2.Use )
   END_RUNG
   RUNG wire#powerrail
      { S7_Templates := "SrcType := Int" } NE_Contact(in1 := "Time_SYS_DB".Time_Now.Minute, in2 := #ON_2."M")
   END_RUNG wire#w1
   // the same network as SCL:
   IF ("Time_SYS_DB".Time_Now.Hour = #ON_2.H) AND ("Time_SYS_DB".Time_Now.Minute = #ON_2."M") THEN
       #ON_2.Use := TRUE;
   END_IF;
   IF ("Time_SYS_DB".Time_Now.Hour <> #ON_2.H) OR ("Time_SYS_DB".Time_Now.Minute <> #ON_2."M") THEN
       #ON_2.Use := FALSE;
   END_IF;
END_REGION

REGION Network 3: Line 1
   RUNG wire#powerrail
      Contact( "pulse_1s" )
      Contact( "Line_Control_DB".Line[1].Start )
      wire#w1
      Div(in1 := "Line_Control_DB".Line[1].Flow, in2 := 3600.0, out => #x0)
      Add(in1 := #Line_1[0].Water, in2 := #x0, out => #Line_1[0].Water)
   END_RUNG
   RUNG wire#w1
      Div(in1 := "Line_Control_DB".Line[1].SP_M, in2 := 60.0, out => #x1)
      Add(in1 := #Line_1[0].Reagent, in2 := #x1, out => #Line_1[0].Reagent)
   END_RUNG
   RUNG wire#powerrail
      P_Contact(operand := #ON_1.Use, bit := #pos[4])
      wire#w2
      Move(in := #Line_1[1].Water, out1 => #Line_1[2].Water)
      Move(in := #Line_1[0].Water, out1 => #Line_1[1].Water)
      Move(in := 0.0, out1 => #Line_1[0].Water)
   END_RUNG
   RUNG wire#powerrail
      P_Contact(operand := #ON_2.Use, bit := #pos[5])
   END_RUNG wire#w2
   RUNG wire#w2
      Move(in := #Line_1[1].Reagent, out1 => #Line_1[2].Reagent)
      Move(in := #Line_1[0].Reagent, out1 => #Line_1[1].Reagent)
      Move(in := 0.0, out1 => #Line_1[0].Reagent)
   END_RUNG
   // the same network as SCL:
   IF "pulse_1s" AND "Line_Control_DB".Line[1].Start THEN
       #x0 := "Line_Control_DB".Line[1].Flow / 3600.0;
       #Line_1[0].Water := #Line_1[0].Water + #x0;
       #x1 := "Line_Control_DB".Line[1].SP_M / 60.0;
       #Line_1[0].Reagent := #Line_1[0].Reagent + #x1;
   END_IF;
   #_w1 := #ON_1.Use AND NOT #pos[4];   // rising edge of #ON_1.Use
   #pos[4] := #ON_1.Use;
   #_w2 := #ON_2.Use AND NOT #pos[5];   // rising edge of #ON_2.Use
   #pos[5] := #ON_2.Use;
   IF #_w1 OR #_w2 THEN
       #Line_1[2].Water := #Line_1[1].Water;
       #Line_1[1].Water := #Line_1[0].Water;
       #Line_1[0].Water := 0.0;
       #Line_1[2].Reagent := #Line_1[1].Reagent;
       #Line_1[1].Reagent := #Line_1[0].Reagent;
       #Line_1[0].Reagent := 0.0;
   END_IF;
END_REGION

REGION Network 4
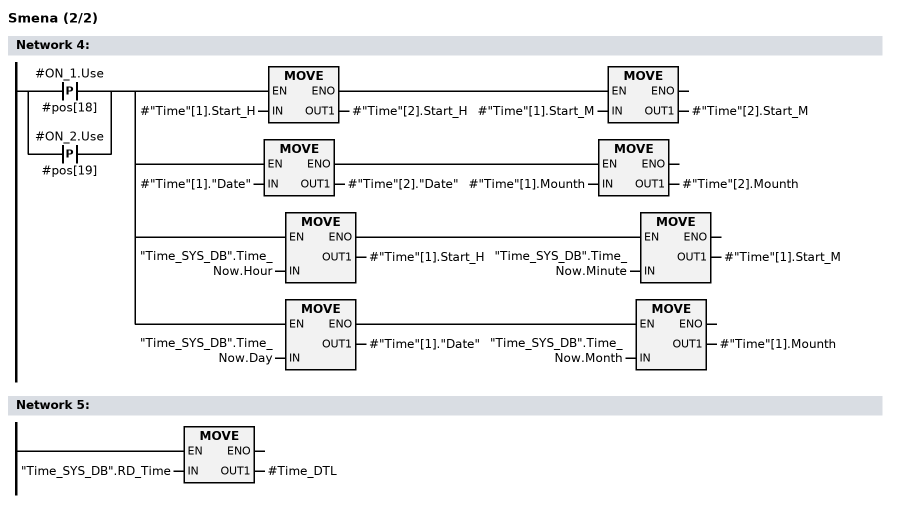
   RUNG wire#powerrail
      P_Contact(operand := #ON_1.Use, bit := #pos[18])
      wire#w1
      Move(in := #"Time"[1].Start_H, out1 => #"Time"[2].Start_H)
      Move(in := #"Time"[1].Start_M, out1 => #"Time"[2].Start_M)
   END_RUNG
   RUNG wire#powerrail
      P_Contact(operand := #ON_2.Use, bit := #pos[19])
   END_RUNG wire#w1
   RUNG wire#w1
      Move(in := #"Time"[1]."Date", out1 => #"Time"[2]."Date")
      Move(in := #"Time"[1].Mounth, out1 => #"Time"[2].Mounth)
   END_RUNG
   RUNG wire#w1
      Move(in := "Time_SYS_DB".Time_Now.Hour, out1 => #"Time"[1].Start_H)
      Move(in := "Time_SYS_DB".Time_Now.Minute, out1 => #"Time"[1].Start_M)
   END_RUNG
   RUNG wire#w1
      Move(in := "Time_SYS_DB".Time_Now.Day, out1 => #"Time"[1]."Date")
      Move(in := "Time_SYS_DB".Time_Now.Month, out1 => #"Time"[1].Mounth)
   END_RUNG
   // the same network as SCL:
   #_w1 := #ON_1.Use AND NOT #pos[18];   // rising edge of #ON_1.Use
   #pos[18] := #ON_1.Use;
   #_w2 := #ON_2.Use AND NOT #pos[19];   // rising edge of #ON_2.Use
   #pos[19] := #ON_2.Use;
   IF #_w1 OR #_w2 THEN
       #"Time"[2].Start_H := #"Time"[1].Start_H;
       #"Time"[2].Start_M := #"Time"[1].Start_M;
       #"Time"[2]."Date" := #"Time"[1]."Date";
       #"Time"[2].Mounth := #"Time"[1].Mounth;
       #"Time"[1].Start_H := "Time_SYS_DB".Time_Now.Hour;
       #"Time"[1].Start_M := "Time_SYS_DB".Time_Now.Minute;
       #"Time"[1]."Date" := "Time_SYS_DB".Time_Now.Day;
       #"Time"[1].Mounth := "Time_SYS_DB".Time_Now.Month;
   END_IF;
END_REGION

REGION Network 5
   RUNG wire#powerrail
      Move(in := "Time_SYS_DB".RD_Time, out1 => #Time_DTL)
   END_RUNG
   // the same network as SCL:
   #Time_DTL := "Time_SYS_DB".RD_Time;
END_REGION
END_FUNCTION_BLOCK

FUNCTION_BLOCK "PIDx"   // FB260, LAD
{ S7_Optimized_Access := 'TRUE' }
VERSION : 0.1
// stored: AutoNumber false, IsIECCheckEnabled false, IsRetainMemResEnabled false, MemoryReserve 100, SetENOAutomatically false, UDAEnableTagReadback false
   VAR DB_SPECIFIC
      Time_DTL { S7_SetPoint := 'True'} : DTL;
   END_VAR
BEGIN

REGION Network 1
